      ;FOLD -- Hilfsflag SK Programmwechsel -- ;%{SE}%MKUKATPVW %CVW_COM %VCOMMENT %P 2:-- Hilfsflag SK Programmwechsel --, 3: VW_COMMENT
      ;ENDFOLD
      ;FOLD F334 = AUS ;%{SE}%MKUKATPVW %CVW_SPS %VBOASG %P 2:F334 = AUS, 3: BOASG
         $FLAG[334] = FALSE
      ;ENDFOLD
      ;FOLD A757 = F830 & A757 ;%{SE}%MKUKATPVW %CVW_SPS %VBOASG %P 2:A757 = F830 & A757, 3: BOASG
         $OUT[757] = $FLAG[830] AND $OUT[757]
      ;ENDFOLD
      ;FOLD -- EZ1/SP1 schliessen -- ;%{SE}%MKUKATPVW %CVW_COM %VCOMMENT %P 2:-- EZ1/SP1 schliessen --, 3: VW_COMMENT
      ;ENDFOLD
      ;FOLD A725 = !F830 & A725 ;%{SE}%MKUKATPVW %CVW_SPS %VBOASG %P 2:A725 = !F830 & A725, 3: BOASG
         $OUT[725] = NOT $FLAG[830] AND $OUT[725]
      ;ENDFOLD
      ;FOLD A717 = AUS ;%{SE}%MKUKATPVW %CVW_SPS %VBOASG %P 2:A717 = AUS, 3: BOASG
         $OUT[717] = FALSE
      ;ENDFOLD
      ;FOLD A718 = !F329 & !F122 ;%{SE}%MKUKATPVW %CVW_SPS %VBOASG %P 2:A718 = !F329 & !F122, 3: BOASG
         $OUT[718] = NOT $FLAG[329] AND NOT $FLAG[122]
      ;ENDFOLD
      ;FOLD -- Ueberwachungszeit Kurzschlussschweissung SK1 -- ;%{SE}%MKUKATPVW %CVW_COM %VCOMMENT %P 2:-- Ueberwachungszeit Kurzschlussschweissung SK1 --, 3: VW_COMMENT
      ;ENDFOLD
      ;FOLD t9 ( EIN ) = -80[1/10Sek] ;%{SE}%MKUKATPVW %CVW_SPS %VTASG %P 2:t9 ( EIN ) = -80[1/10Sek], 3: TASG
         VW(#SET_TIME,TRUE,9,0,-80)
      ;ENDFOLD
      ;FOLD Schritt 71 = T8 & !E717 & E718 + E717 & !E718 & (F329 + F326 + F122) & A4039  ;%{SE}%MKUKATPVW %CVW_SPS %VST_CON %P 2:Schritt 71 = T8 & !E717 & E718 + E717 & !E718 & (F329 + F326 + F122) & A4039 , 3: ST_CON
         IF $TIMER_FLAG[8] AND NOT $IN[717] AND $IN[718] OR $IN[717] AND NOT $IN[718] AND ($FLAG[329] OR $FLAG[326] OR $FLAG[122]) AND $OUT[4039] THEN
            PREVSTEP = $APP_INT[5]
            $APP_INT[5] = 71
         ENDIF
      ;ENDFOLD
   ;ENDFOLD
   ;FOLD SCHRITT 71 -- STAT EZ1/SP1/KE1-- ;%{P}%MKUKATPVW,%CSTEP,%VST_NR,%P 1:SCHRITT, 2:71, 3: STAT EZ1/SP1/KE1
      ;FOLD ;%{H}
         Case 71
      ;ENDFOLD
      ;FOLD -- Hilfsflag SK Programmwechsel -- ;%{SE}%MKUKATPVW %CVW_COM %VCOMMENT %P 2:-- Hilfsflag SK Programmwechsel --, 3: VW_COMMENT
      ;ENDFOLD
      ;FOLD F334 = AUS ;%{SE}%MKUKATPVW %CVW_SPS %VBOASG %P 2:F334 = AUS, 3: BOASG
         $FLAG[334] = FALSE
      ;ENDFOLD
      ;FOLD t9 ( EIN ) = STOP ;%{SE}%MKUKATPVW %CVW_SPS %VTSTOP %P 2:t9 ( EIN ) = STOP, 3: TSTOP
         VW(#SET_TIME,TRUE,9,1,0)
      ;ENDFOLD
      ;FOLD -- RSK Fehlerausgabe Kraftaufbau -- ;%{SE}%MKUKATPVW %CVW_COM %VCOMMENT %P 2:-- RSK Fehlerausgabe Kraftaufbau --, 3: VW_COMMENT
      ;ENDFOLD
      ;FOLD F325 = T9 + F325 ;%{SE}%MKUKATPVW %CVW_SPS %VBOASG %P 2:F325 = T9 + F325, 3: BOASG
         $FLAG[325] = $TIMER_FLAG[9] OR $FLAG[325]
      ;ENDFOLD
      ;FOLD -- RSK Fehlerausgabe K -- ;%{SE}%MKUKATPVW %CVW_COM %VCOMMENT %P 2:-- RSK Fehlerausgabe K --, 3: VW_COMMENT
      ;ENDFOLD
      ;FOLD F836 = (A718 & E788 + A718 & !E705) & F830 ;%{SE}%MKUKATPVW %CVW_SPS %VBOASG %P 2:F836 = (A718 & E788 + A718 & !E705) & F830, 3: BOASG
         $FLAG[836] = ($OUT[718] AND $IN[788] OR $OUT[718] AND NOT $IN[705]) AND $FLAG[830]
      ;ENDFOLD
      ;FOLD F327 = (A785 & E805 + A785 & !E802) &!F830 + F836 + F327 ;%{SE}%MKUKATPVW %CVW_SPS %VBOASG %P 2:F327 = (A785 & E805 + A785 & !E802) &!F830 + F836 + F327, 3: BOASG
         $FLAG[327] = ($OUT[785] AND $IN[805] OR $OUT[785] AND NOT $IN[802]) AND NOT $FLAG[830] OR $FLAG[836] OR $FLAG[327]
      ;ENDFOLD
      ;FOLD -- RSK Sammelstoerung -- ;%{SE}%MKUKATPVW %CVW_COM %VCOMMENT %P 2:-- RSK Sammelstoerung --, 3: VW_COMMENT
      ;ENDFOLD
      ;FOLD F329 = F325 + F326 + F327 ;%{SE}%MKUKATPVW %CVW_SPS %VBOASG %P 2:F329 = F325 + F326 + F327, 3: BOASG
         $FLAG[329] = $FLAG[325] OR $FLAG[326] OR $FLAG[327]
      ;ENDFOLD
      ;FOLD -- Kurzschlussschweissung SK1 -- ;%{SE}%MKUKATPVW %CVW_COM %VCOMMENT %P 2:-- Kurzschlussschweissung SK1 --, 3: VW_COMMENT
      ;ENDFOLD
      ;FOLD A785 = (!F325 & !F329 & !F122 & !F830) + (F830 & A785) ;%{SE}%MKUKATPVW %CVW_SPS %VBOASG %P 2:A785 = (!F325 & !F329 & !F122 & !F830) + (F830 & A785), 3: BOASG
         $OUT[785] = (NOT $FLAG[325] AND NOT $FLAG[329] AND NOT $FLAG[122] AND NOT $FLAG[830]) OR ($FLAG[830] AND $OUT[785])
      ;ENDFOLD
      ;FOLD F836 = AUS ;%{SE}%MKUKATPVW %CVW_SPS %VBOASG %P 2:F836 = AUS, 3: BOASG
         $FLAG[836] = FALSE
      ;ENDFOLD
      ;FOLD F836 = (E719 & E787 & !E789 + E719 & E15 + F326 + F327 + F122) & F830 & A4039 ;%{SE}%MKUKATPVW %CVW_SPS %VBOASG %P 2:F836 = (E719 & E787 & !E789 + E719 & E15 + F326 + F327 + F122) & F830 & A4039, 3: BOASG
         $FLAG[836] = ($IN[719] AND $IN[787] AND NOT $IN[789] OR $IN[719] AND $IN[15] OR $FLAG[326] OR $FLAG[327] OR $FLAG[122]) AND $FLAG[830] AND $OUT[4039]
      ;ENDFOLD
      ;FOLD -- Flagbildung Wiederholfraesen -- ;%{SE}%MKUKATPVW %CVW_COM %VCOMMENT %P 2:-- Flagbildung Wiederholfraesen --, 3: VW_COMMENT
      ;ENDFOLD
      ;FOLD F749 = (F322 + F323 + F325 + F326 + F327 + F329) & !F748 ;%{SE}%MKUKATPVW %CVW_SPS %VBOASG %P 2:F749 = (F322 + F323 + F325 + F326 + F327 + F329) & !F748, 3: BOASG
         $FLAG[749] = ($FLAG[322] OR $FLAG[323] OR $FLAG[325] OR $FLAG[326] OR $FLAG[327] OR $FLAG[329]) AND NOT $FLAG[748]
      ;ENDFOLD
      ;FOLD Schritt 72 = (E785 & E804 & !E806 + E785 & E15 + F326 + F327 + F122) & !F830 & A4039 + F836  ;%{SE}%MKUKATPVW %CVW_SPS %VST_CON %P 2:Schritt 72 = (E785 & E804 & !E806 + E785 & E15 + F326 + F327 + F122) & !F830 & A4039 + F836 , 3: ST_CON
         IF ($IN[785] AND $IN[804] AND NOT $IN[806] OR $IN[785] AND $IN[15] OR $FLAG[326] OR $FLAG[327] OR $FLAG[122]) AND NOT $FLAG[830] AND $OUT[4039] OR $FLAG[836] THEN
            PREVSTEP = $APP_INT[5]
            $APP_INT[5] = 72
         ENDIF
      ;ENDFOLD
   ;ENDFOLD
   ;FOLD SCHRITT 72 -- STAT EZ1/SP1/KE1 -- ;%{P}%MKUKATPVW,%CSTEP,%VST_NR,%P 1:SCHRITT, 2:72, 3: STAT EZ1/SP1/KE1
      ;FOLD ;%{H}
         Case 72
      ;ENDFOLD
      ;FOLD A785 = F830 & A785 ;%{SE}%MKUKATPVW %CVW_SPS %VBOASG %P 2:A785 = F830 & A785, 3: BOASG
         $OUT[785] = $FLAG[830] AND $OUT[785]
      ;ENDFOLD
      ;FOLD F78 = !F327 & F78 ;%{SE}%MKUKATPVW %CVW_SPS %VBOASG %P 2:F78 = !F327 & F78, 3: BOASG
         $FLAG[78] = NOT $FLAG[327] AND $FLAG[78]
      ;ENDFOLD
      ;FOLD F79 = F327 + F79 ;%{SE}%MKUKATPVW %CVW_SPS %VBOASG %P 2:F79 = F327 + F79, 3: BOASG
         $FLAG[79] = $FLAG[327] OR $FLAG[79]
      ;ENDFOLD
      ;FOLD F836 = AUS ;%{SE}%MKUKATPVW %CVW_SPS %VBOASG %P 2:F836 = AUS, 3: BOASG
         $FLAG[836] = FALSE
      ;ENDFOLD
      ;FOLD -- EZ1/SP1/KE1 SZ1 oeffnen -- ;%{SE}%MKUKATPVW %CVW_COM %VCOMMENT %P 2:-- EZ1/SP1/KE1 SZ1 oeffnen --, 3: VW_COMMENT
      ;ENDFOLD
      ;FOLD A719 = AUS ;%{SE}%MKUKATPVW %CVW_SPS %VBOASG %P 2:A719 = AUS, 3: BOASG
         $OUT[719] = FALSE
      ;ENDFOLD
      ;FOLD A718 = AUS ;%{SE}%MKUKATPVW %CVW_SPS %VBOASG %P 2:A718 = AUS, 3: BOASG
         $OUT[718] = FALSE
      ;ENDFOLD
      ;FOLD A717 = !E717 ;%{SE}%MKUKATPVW %CVW_SPS %VBOASG %P 2:A717 = !E717, 3: BOASG
         $OUT[717] = NOT $IN[717]
      ;ENDFOLD
      ;FOLD F836 = !F326 & !F830 ;%{SE}%MKUKATPVW %CVW_SPS %VBOASG %P 2:F836 = !F326 & !F830, 3: BOASG
         $FLAG[836] = NOT $FLAG[326] AND NOT $FLAG[830]
      ;ENDFOLD
      ;FOLD bin3 ( F836 ) = 1 ;%{SE}%MKUKATPVW %CVW_SPS %VARIASG %P 2:bin3 ( F836 ) = 1, 3: ARIASG
         VW(#BINOUT,$FLAG[836],3,1)
      ;ENDFOLD
      ;FOLD -- Wartezeit Programmwechsel SK -- ;%{SE}%MKUKATPVW %CVW_COM %VCOMMENT %P 2:-- Wartezeit Programmwechsel SK --, 3: VW_COMMENT
      ;ENDFOLD
      ;FOLD T8 ( !F334 ) = -2[1/10Sek] ;%{SE}%MKUKATPVW %CVW_SPS %VTASG %P 2:T8 ( !F334 ) = -2[1/10Sek], 3: TASG
         VW(#SET_TIME,NOT $FLAG[334],8,0,-2)
      ;ENDFOLD
      ;FOLD -- Hilfsflag SK Programmwechsel -- ;%{SE}%MKUKATPVW %CVW_COM %VCOMMENT %P 2:-- Hilfsflag SK Programmwechsel --, 3: VW_COMMENT
      ;ENDFOLD
      ;FOLD F334 = EIN ;%{SE}%MKUKATPVW %CVW_SPS %VBOASG %P 2:F334 = EIN, 3: BOASG
         $FLAG[334] = TRUE
      ;ENDFOLD
      ;FOLD F748 = F322 + F323 + F325 + F326 + F327 + F329 ;%{SE}%MKUKATPVW %CVW_SPS %VBOASG %P 2:F748 = F322 + F323 + F325 + F326 + F327 + F329, 3: BOASG
         $FLAG[748] = $FLAG[322] OR $FLAG[323] OR $FLAG[325] OR $FLAG[326] OR $FLAG[327] OR $FLAG[329]
      ;ENDFOLD
      ;FOLD Schritt 51 = E717 & !E718 & (F322 + F323 + F325 + F326 + F327 + F329) & (E26 + E27) & A4039  ;%{SE}%MKUKATPVW %CVW_SPS %VST_CON %P 2:Schritt 51 = E717 & !E718 & (F322 + F323 + F325 + F326 + F327 + F329) & (E26 + E27) & A4039 , 3: ST_CON
         IF $IN[717] AND NOT $IN[718] AND ($FLAG[322] OR $FLAG[323] OR $FLAG[325] OR $FLAG[326] OR $FLAG[327] OR $FLAG[329]) AND ($IN[26] OR $IN[27]) AND $OUT[4039] THEN
            PREVSTEP = $APP_INT[5]
            $APP_INT[5] = 51
         ENDIF
      ;ENDFOLD
      ;FOLD Schritt 51 = E717 & !E718 & (F322 + F323 + F325 + F326 + F327 + F329) & (F749 & F731) & A4039  ;%{SE}%MKUKATPVW %CVW_SPS %VST_CON %P 2:Schritt 51 = E717 & !E718 & (F322 + F323 + F325 + F326 + F327 + F329) & (F749 & F731) & A4039 , 3: ST_CON
         IF $IN[717] AND NOT $IN[718] AND ($FLAG[322] OR $FLAG[323] OR $FLAG[325] OR $FLAG[326] OR $FLAG[327] OR $FLAG[329]) AND ($FLAG[749] AND $FLAG[731]) AND $OUT[4039] THEN
            PREVSTEP = $APP_INT[5]
            $APP_INT[5] = 51
         ENDIF
      ;ENDFOLD
      ;FOLD Schritt 73 = T8 & E717 & !E718 & (!F325 & !F326 & !F327 & !F329 + F122) & A4039  ;%{SE}%MKUKATPVW %CVW_SPS %VST_CON %P 2:Schritt 73 = T8 & E717 & !E718 & (!F325 & !F326 & !F327 & !F329 + F122) & A4039 , 3: ST_CON
         IF $TIMER_FLAG[8] AND $IN[717] AND NOT $IN[718] AND (NOT $FLAG[325] AND NOT $FLAG[326] AND NOT $FLAG[327] AND NOT $FLAG[329] OR $FLAG[122]) AND $OUT[4039] THEN
            PREVSTEP = $APP_INT[5]
            $APP_INT[5] = 73
         ENDIF
      ;ENDFOLD
   ;ENDFOLD
   ;FOLD SCHRITT 73 -- STAT EZ1/SP1/KE1 # Ende -- ;%{P}%MKUKATPVW,%CSTEP,%VST_NR,%P 1:SCHRITT, 2:73, 3: STAT EZ1/SP1/KE1 # Ende
      ;FOLD ;%{H}
         Case 73
      ;ENDFOLD
      ;FOLD -- Hilfsflag SK Programmwechsel -- ;%{SE}%MKUKATPVW %CVW_COM %VCOMMENT %P 2:-- Hilfsflag SK Programmwechsel --, 3: VW_COMMENT
      ;ENDFOLD
      ;FOLD F334 = AUS ;%{SE}%MKUKATPVW %CVW_SPS %VBOASG %P 2:F334 = AUS, 3: BOASG
         $FLAG[334] = FALSE
      ;ENDFOLD
      ;FOLD A116 = AUS ;%{SE}%MKUKATPVW %CVW_SPS %VBOASG %P 2:A116 = AUS, 3: BOASG
         $OUT[116] = FALSE
      ;ENDFOLD
      ;FOLD A130 = AUS ;%{SE}%MKUKATPVW %CVW_SPS %VBOASG %P 2:A130 = AUS, 3: BOASG
         $OUT[130] = FALSE
      ;ENDFOLD
      ;FOLD F836 = AUS ;%{SE}%MKUKATPVW %CVW_SPS %VBOASG %P 2:F836 = AUS, 3: BOASG
         $FLAG[836] = FALSE
      ;ENDFOLD
      ;FOLD -- RSK Sammelstoerung -- ;%{SE}%MKUKATPVW %CVW_COM %VCOMMENT %P 2:-- RSK Sammelstoerung --, 3: VW_COMMENT
      ;ENDFOLD
      ;FOLD F329 = F122 ;%{SE}%MKUKATPVW %CVW_SPS %VBOASG %P 2:F329 = F122, 3: BOASG
         $FLAG[329] = $FLAG[122]
      ;ENDFOLD
      ;FOLD F93 = (!E786 & E787 & !E788 & !F830) + (!E721 & !E723 & E724 & F830) + F122 & (E26 + E27) ;%{SE}%MKUKATPVW %CVW_SPS %VBOASG %P 2:F93 = (!E786 & E787 & !E788 & !F830) + (!E721 & !E723 & E724 & F830) + F122 & (E26 + E27), 3: BOASG
         $FLAG[93] = (NOT $IN[786] AND $IN[787] AND NOT $IN[788] AND NOT $FLAG[830]) OR (NOT $IN[721] AND NOT $IN[723] AND $IN[724] AND $FLAG[830]) OR $FLAG[122] AND ($IN[26] OR $IN[27])
      ;ENDFOLD
      ;FOLD Schritt 1 = F93 & A4039  ;%{SE}%MKUKATPVW %CVW_SPS %VST_CON %P 2:Schritt 1 = F93 & A4039 , 3: ST_CON
         IF $FLAG[93] AND $OUT[4039] THEN
            PREVSTEP = $APP_INT[5]
            $APP_INT[5] = 1
         ENDIF
      ;ENDFOLD
   ;ENDFOLD
   ;FOLD SCHRITT 74 -- STAT EZ2/SP2/KE2 # Start-- ;%{P}%MKUKATPVW,%CSTEP,%VST_NR,%P 1:SCHRITT, 2:74, 3: STAT EZ2/SP2/KE2 # Start
      ;FOLD ;%{H}
         Case 74
      ;ENDFOLD
      ;FOLD -- RSK gestartet -- ;%{SE}%MKUKATPVW %CVW_COM %VCOMMENT %P 2:-- RSK gestartet --, 3: VW_COMMENT
      ;ENDFOLD
      ;FOLD F160 = AUS ;%{SE}%MKUKATPVW %CVW_SPS %VBOASG %P 2:F160 = AUS, 3: BOASG
         $FLAG[160] = FALSE
      ;ENDFOLD
      ;FOLD F321 = AUS ;%{SE}%MKUKATPVW %CVW_SPS %VBOASG %P 2:F321 = AUS, 3: BOASG
         $FLAG[321] = FALSE
      ;ENDFOLD
      ;FOLD F322 = AUS ;%{SE}%MKUKATPVW %CVW_SPS %VBOASG %P 2:F322 = AUS, 3: BOASG
         $FLAG[322] = FALSE
      ;ENDFOLD
      ;FOLD F323 = AUS ;%{SE}%MKUKATPVW %CVW_SPS %VBOASG %P 2:F323 = AUS, 3: BOASG
         $FLAG[323] = FALSE
      ;ENDFOLD
      ;FOLD F324 = AUS ;%{SE}%MKUKATPVW %CVW_SPS %VBOASG %P 2:F324 = AUS, 3: BOASG
         $FLAG[324] = FALSE
      ;ENDFOLD
      ;FOLD F325 = AUS ;%{SE}%MKUKATPVW %CVW_SPS %VBOASG %P 2:F325 = AUS, 3: BOASG
         $FLAG[325] = FALSE
      ;ENDFOLD
      ;FOLD F326 = AUS ;%{SE}%MKUKATPVW %CVW_SPS %VBOASG %P 2:F326 = AUS, 3: BOASG
         $FLAG[326] = FALSE
      ;ENDFOLD
      ;FOLD F327 = AUS ;%{SE}%MKUKATPVW %CVW_SPS %VBOASG %P 2:F327 = AUS, 3: BOASG
         $FLAG[327] = FALSE
      ;ENDFOLD
      ;FOLD F329 = AUS ;%{SE}%MKUKATPVW %CVW_SPS %VBOASG %P 2:F329 = AUS, 3: BOASG
         $FLAG[329] = FALSE
      ;ENDFOLD
      ;FOLD -- EZ2/SP2/KE2 Zaehler -- ;%{SE}%MKUKATPVW %CVW_COM %VCOMMENT %P 2:-- EZ2/SP2/KE2 Zaehler --, 3: VW_COMMENT
      ;ENDFOLD
      ;FOLD F150 = AUS ;%{SE}%MKUKATPVW %CVW_SPS %VBOASG %P 2:F150 = AUS, 3: BOASG
         $FLAG[150] = FALSE
      ;ENDFOLD
      ;FOLD F151 = AUS ;%{SE}%MKUKATPVW %CVW_SPS %VBOASG %P 2:F151 = AUS, 3: BOASG
         $FLAG[151] = FALSE
      ;ENDFOLD
      ;FOLD F152 = AUS ;%{SE}%MKUKATPVW %CVW_SPS %VBOASG %P 2:F152 = AUS, 3: BOASG
         $FLAG[152] = FALSE
      ;ENDFOLD
      ;FOLD F153 = AUS ;%{SE}%MKUKATPVW %CVW_SPS %VBOASG %P 2:F153 = AUS, 3: BOASG
         $FLAG[153] = FALSE
      ;ENDFOLD
      ;FOLD F154 = AUS ;%{SE}%MKUKATPVW %CVW_SPS %VBOASG %P 2:F154 = AUS, 3: BOASG
         $FLAG[154] = FALSE
      ;ENDFOLD
      ;FOLD F155 = AUS ;%{SE}%MKUKATPVW %CVW_SPS %VBOASG %P 2:F155 = AUS, 3: BOASG
         $FLAG[155] = FALSE
      ;ENDFOLD
      ;FOLD -- Hilfsflags Funktionstest KF Motor -- ;%{SE}%MKUKATPVW %CVW_COM %VCOMMENT %P 2:-- Hilfsflags Funktionstest KF Motor --, 3: VW_COMMENT
      ;ENDFOLD
      ;FOLD F312 = AUS ;%{SE}%MKUKATPVW %CVW_SPS %VBOASG %P 2:F312 = AUS, 3: BOASG
         $FLAG[312] = FALSE
      ;ENDFOLD
      ;FOLD F313 = AUS ;%{SE}%MKUKATPVW %CVW_SPS %VBOASG %P 2:F313 = AUS, 3: BOASG
         $FLAG[313] = FALSE
      ;ENDFOLD
      ;FOLD bin3 ( F285 ) = 35 ;%{SE}%MKUKATPVW %CVW_SPS %VARIASG %P 2:bin3 ( F285 ) = 35, 3: ARIASG
         VW(#BINOUT,$FLAG[285],3,35)
      ;ENDFOLD
      ;FOLD bin4 ( EIN ) = 31 ;%{SE}%MKUKATPVW %CVW_SPS %VARIASG %P 2:bin4 ( EIN ) = 31, 3: ARIASG
         VW(#BINOUT,TRUE,4,31)
      ;ENDFOLD
      ;FOLD bin6 ( !F285 ) = 31 ;%{SE}%MKUKATPVW %CVW_SPS %VARIASG %P 2:bin6 ( !F285 ) = 31, 3: ARIASG
         VW(#BINOUT,NOT $FLAG[285],6,31)
      ;ENDFOLD
      ;FOLD -- Wartezeit Programmwechsel SK -- ;%{SE}%MKUKATPVW %CVW_COM %VCOMMENT %P 2:-- Wartezeit Programmwechsel SK --, 3: VW_COMMENT
      ;ENDFOLD
      ;FOLD T8 ( !F334 ) = -2[1/10Sek] ;%{SE}%MKUKATPVW %CVW_SPS %VTASG %P 2:T8 ( !F334 ) = -2[1/10Sek], 3: TASG
         VW(#SET_TIME,NOT $FLAG[334],8,0,-2)
      ;ENDFOLD
      ;FOLD -- Hilfsflag SK Programmwechsel -- ;%{SE}%MKUKATPVW %CVW_COM %VCOMMENT %P 2:-- Hilfsflag SK Programmwechsel --, 3: VW_COMMENT
      ;ENDFOLD
      ;FOLD F334 = EIN ;%{SE}%MKUKATPVW %CVW_SPS %VBOASG %P 2:F334 = EIN, 3: BOASG
         $FLAG[334] = TRUE
      ;ENDFOLD
      ;FOLD -- Stat. EZ2/SP2/KE2 beim Fraesen -- ;%{SE}%MKUKATPVW %CVW_COM %VCOMMENT %P 2:-- Stat. EZ2/SP2/KE2 beim Fraesen --, 3: VW_COMMENT
      ;ENDFOLD
      ;FOLD A116 = EIN ;%{SE}%MKUKATPVW %CVW_SPS %VBOASG %P 2:A116 = EIN, 3: BOASG
         $OUT[116] = TRUE
      ;ENDFOLD
      ;FOLD A162 = EIN ;%{SE}%MKUKATPVW %CVW_SPS %VBOASG %P 2:A162 = EIN, 3: BOASG
         $OUT[162] = TRUE
      ;ENDFOLD
      ;FOLD -- Quitt. Fraesen SK1 AUS -- ;%{SE}%MKUKATPVW %CVW_COM %VCOMMENT %P 2:-- Quitt. Fraesen SK1 AUS --, 3: VW_COMMENT
      ;ENDFOLD
      ;FOLD A786 = F830 ;%{SE}%MKUKATPVW %CVW_SPS %VBOASG %P 2:A786 = F830, 3: BOASG
         $OUT[786] = $FLAG[830]
      ;ENDFOLD
      ;FOLD A722 = !F830 ;%{SE}%MKUKATPVW %CVW_SPS %VBOASG %P 2:A722 = !F830, 3: BOASG
         $OUT[722] = NOT $FLAG[830]
      ;ENDFOLD
      ;FOLD -- Quitt. Fraesen SK2 AUS -- ;%{SE}%MKUKATPVW %CVW_COM %VCOMMENT %P 2:-- Quitt. Fraesen SK2 AUS --, 3: VW_COMMENT
      ;ENDFOLD
      ;FOLD A946 = F831 & A946 ;%{SE}%MKUKATPVW %CVW_SPS %VBOASG %P 2:A946 = F831 & A946, 3: BOASG
         $OUT[946] = $FLAG[831] AND $OUT[946]
      ;ENDFOLD
      ;FOLD A882 = !F831 & A882 ;%{SE}%MKUKATPVW %CVW_SPS %VBOASG %P 2:A882 = !F831 & A882, 3: BOASG
         $OUT[882] = NOT $FLAG[831] AND $OUT[882]
      ;ENDFOLD
      ;FOLD Schritt 75 = T8 & A4039  ;%{SE}%MKUKATPVW %CVW_SPS %VST_CON %P 2:Schritt 75 = T8 & A4039 , 3: ST_CON
         IF $TIMER_FLAG[8] AND $OUT[4039] THEN
            PREVSTEP = $APP_INT[5]
            $APP_INT[5] = 75
         ENDIF
      ;ENDFOLD
   ;ENDFOLD
   ;FOLD SCHRITT 75 -- STAT EZ2/SP2/KE2 -- ;%{P}%MKUKATPVW,%CSTEP,%VST_NR,%P 1:SCHRITT, 2:75, 3: STAT EZ2/SP2/KE2
      ;FOLD ;%{H}
         Case 75
      ;ENDFOLD
      ;FOLD -- Hilfsflag SK Programmwechsel -- ;%{SE}%MKUKATPVW %CVW_COM %VCOMMENT %P 2:-- Hilfsflag SK Programmwechsel --, 3: VW_COMMENT
      ;ENDFOLD
      ;FOLD F334 = AUS ;%{SE}%MKUKATPVW %CVW_SPS %VBOASG %P 2:F334 = AUS, 3: BOASG
         $FLAG[334] = FALSE
      ;ENDFOLD
      ;FOLD -- Ueberwachungszeit KF2 EIN -- ;%{SE}%MKUKATPVW %CVW_COM %VCOMMENT %P 2:-- Ueberwachungszeit KF2 EIN --, 3: VW_COMMENT
      ;ENDFOLD
      ;FOLD T7 ( EIN ) = -50[1/10Sek] ;%{SE}%MKUKATPVW %CVW_SPS %VTASG %P 2:T7 ( EIN ) = -50[1/10Sek], 3: TASG
         VW(#SET_TIME,TRUE,7,0,-50)
      ;ENDFOLD
      ;FOLD -- KF2 einschalten -- ;%{SE}%MKUKATPVW %CVW_COM %VCOMMENT %P 2:-- KF2 einschalten --, 3: VW_COMMENT
      ;ENDFOLD
      ;FOLD i1 (EIN) = 0 ;%{SE}%MKUKATPVW %CVW_SPS %VARIASG %P 2:i1 (EIN) = 0, 3: ARIASG
         VW(#COUNTER,TRUE,1,0)
      ;ENDFOLD
      ;FOLD A994 = EIN ;%{SE}%MKUKATPVW %CVW_SPS %VBOASG %P 2:A994 = EIN, 3: BOASG
         $OUT[994] = TRUE
      ;ENDFOLD
      ;FOLD Schritt 76 = A4039  ;%{SE}%MKUKATPVW %CVW_SPS %VST_CON %P 2:Schritt 76 = A4039 , 3: ST_CON
         IF $OUT[4039] THEN
            PREVSTEP = $APP_INT[5]
            $APP_INT[5] = 76
         ENDIF
      ;ENDFOLD
   ;ENDFOLD
   ;FOLD SCHRITT 76 -- STAT EZ2/SP2/KE2 -- ;%{P}%MKUKATPVW,%CSTEP,%VST_NR,%P 1:SCHRITT, 2:76, 3: STAT EZ2/SP2/KE2
      ;FOLD ;%{H}
         Case 76
      ;ENDFOLD
      ;FOLD -- Funktionstest KF Motor -- ;%{SE}%MKUKATPVW %CVW_COM %VCOMMENT %P 2:-- Funktionstest KF Motor --, 3: VW_COMMENT
      ;ENDFOLD
      ;FOLD F312 = EIN ;%{SE}%MKUKATPVW %CVW_SPS %VBOASG %P 2:F312 = EIN, 3: BOASG
         $FLAG[312] = TRUE
      ;ENDFOLD
      ;FOLD F313 = i1 > 2 ;%{SE}%MKUKATPVW %CVW_SPS %VBOCMP %P 2:F313 = i1 > 2, 3: BOCMP
         $FLAG[313] = $COUNT_I[1] > 2
      ;ENDFOLD
      ;FOLD Schritt 77 = (F313 + T7) & A4039  ;%{SE}%MKUKATPVW %CVW_SPS %VST_CON %P 2:Schritt 77 = (F313 + T7) & A4039 , 3: ST_CON
         IF ($FLAG[313] OR $TIMER_FLAG[7]) AND $OUT[4039] THEN
            PREVSTEP = $APP_INT[5]
            $APP_INT[5] = 77
         ENDIF
      ;ENDFOLD
   ;ENDFOLD
   ;FOLD SCHRITT 77 -- STAT EZ2/SP2/KE2-- ;%{P}%MKUKATPVW,%CSTEP,%VST_NR,%P 1:SCHRITT, 2:77, 3: STAT EZ2/SP2/KE2
      ;FOLD ;%{H}
         Case 77
      ;ENDFOLD
      ;FOLD F312 = AUS ;%{SE}%MKUKATPVW %CVW_SPS %VBOASG %P 2:F312 = AUS, 3: BOASG
         $FLAG[312] = FALSE
      ;ENDFOLD
      ;FOLD -- Ueberwachungszeit KS2 schwenken -- ;%{SE}%MKUKATPVW %CVW_COM %VCOMMENT %P 2:-- Ueberwachungszeit KS2 schwenken --, 3: VW_COMMENT
      ;ENDFOLD
      ;FOLD t8 ( EIN ) = -100[1/10Sek] ;%{SE}%MKUKATPVW %CVW_SPS %VTASG %P 2:t8 ( EIN ) = -100[1/10Sek], 3: TASG
         VW(#SET_TIME,TRUE,8,0,-100)
      ;ENDFOLD
      ;FOLD Schritt 78 = A4039  ;%{SE}%MKUKATPVW %CVW_SPS %VST_CON %P 2:Schritt 78 = A4039 , 3: ST_CON
         IF $OUT[4039] THEN
            PREVSTEP = $APP_INT[5]
            $APP_INT[5] = 78
         ENDIF
      ;ENDFOLD
   ;ENDFOLD
   ;FOLD SCHRITT 78 -- STAT EZ2/SP2/KE2 -- ;%{P}%MKUKATPVW,%CSTEP,%VST_NR,%P 1:SCHRITT, 2:78, 3: STAT EZ2/SP2/KE2
      ;FOLD ;%{H}
         Case 78
      ;ENDFOLD
      ;FOLD -- RSK Fehlerausgabe KF1 Initiator/Motor -- ;%{SE}%MKUKATPVW %CVW_COM %VCOMMENT %P 2:-- RSK Fehlerausgabe KF1 Initiator/Motor --, 3: VW_COMMENT
      ;ENDFOLD
      ;FOLD F322 = !F313 ;%{SE}%MKUKATPVW %CVW_SPS %VBOASG %P 2:F322 = !F313, 3: BOASG
         $FLAG[322] = NOT $FLAG[313]
      ;ENDFOLD
      ;FOLD -- RSK Fehlerausgabe KS2 Ruhest. -- ;%{SE}%MKUKATPVW %CVW_COM %VCOMMENT %P 2:-- RSK Fehlerausgabe KS2 Ruhest. --, 3: VW_COMMENT
      ;ENDFOLD
      ;FOLD F323 = (!E1002 + E1003 + E1004 + !E1005) & !F324 & !F328 ;%{SE}%MKUKATPVW %CVW_SPS %VBOASG %P 2:F323 = (!E1002 + E1003 + E1004 + !E1005) & !F324 & !F328, 3: BOASG
         $FLAG[323] = (NOT $IN[1002] OR $IN[1003] OR $IN[1004] OR NOT $IN[1005]) AND NOT $FLAG[324] AND NOT $FLAG[328]
      ;ENDFOLD
      ;FOLD -- RSK Sammelstoerung -- ;%{SE}%MKUKATPVW %CVW_COM %VCOMMENT %P 2:-- RSK Sammelstoerung --, 3: VW_COMMENT
      ;ENDFOLD
      ;FOLD F329 = F322 + F323 ;%{SE}%MKUKATPVW %CVW_SPS %VBOASG %P 2:F329 = F322 + F323, 3: BOASG
         $FLAG[329] = $FLAG[322] OR $FLAG[323]
      ;ENDFOLD
      ;FOLD T7 ( EIN ) = STOP ;%{SE}%MKUKATPVW %CVW_SPS %VTSTOP %P 2:T7 ( EIN ) = STOP, 3: TSTOP
         VW(#SET_TIME,TRUE,7,1,0)
      ;ENDFOLD
      ;FOLD A994 = !F322 & !F323 ;%{SE}%MKUKATPVW %CVW_SPS %VBOASG %P 2:A994 = !F322 & !F323, 3: BOASG
         $OUT[994] = NOT $FLAG[322] AND NOT $FLAG[323]
      ;ENDFOLD
      ;FOLD -- KF2 Versetzeinheit vor -- ;%{SE}%MKUKATPVW %CVW_COM %VCOMMENT %P 2:-- KF2 Versetzeinheit vor --, 3: VW_COMMENT
      ;ENDFOLD
      ;FOLD A995 = !F322 & !F323 & F564 ;%{SE}%MKUKATPVW %CVW_SPS %VBOASG %P 2:A995 = !F322 & !F323 & F564, 3: BOASG
         $OUT[995] = NOT $FLAG[322] AND NOT $FLAG[323] AND $FLAG[564]
      ;ENDFOLD
      ;FOLD Schritt 79 = (!F322 & !F323 & (E995 & F564 + !E995 & !F564) + T8) & A4039  ;%{SE}%MKUKATPVW %CVW_SPS %VST_CON %P 2:Schritt 79 = (!F322 & !F323 & (E995 & F564 + !E995 & !F564) + T8) & A4039 , 3: ST_CON
         IF (NOT $FLAG[322] AND NOT $FLAG[323] AND ($IN[995] AND $FLAG[564] OR NOT $IN[995] AND NOT $FLAG[564]) OR $TIMER_FLAG[8]) AND $OUT[4039] THEN
            PREVSTEP = $APP_INT[5]
            $APP_INT[5] = 79
         ENDIF
      ;ENDFOLD
      ;FOLD Schritt 95 = (F322 + F323) & !F324 & !F328 & A4039  ;%{SE}%MKUKATPVW %CVW_SPS %VST_CON %P 2:Schritt 95 = (F322 + F323) & !F324 & !F328 & A4039 , 3: ST_CON
         IF ($FLAG[322] OR $FLAG[323]) AND NOT $FLAG[324] AND NOT $FLAG[328] AND $OUT[4039] THEN
            PREVSTEP = $APP_INT[5]
            $APP_INT[5] = 95
         ENDIF
      ;ENDFOLD
   ;ENDFOLD
   ;FOLD SCHRITT 79 -- STAT EZ2/SP2/KE2 -- ;%{P}%MKUKATPVW,%CSTEP,%VST_NR,%P 1:SCHRITT, 2:79, 3: STAT EZ2/SP2/KE2
      ;FOLD ;%{H}
         Case 79
      ;ENDFOLD
      ;FOLD -- RSK Sammelstoerung -- ;%{SE}%MKUKATPVW %CVW_COM %VCOMMENT %P 2:-- RSK Sammelstoerung --, 3: VW_COMMENT
      ;ENDFOLD
      ;FOLD F329 = T8 ;%{SE}%MKUKATPVW %CVW_SPS %VBOASG %P 2:F329 = T8, 3: BOASG
         $FLAG[329] = $TIMER_FLAG[8]
      ;ENDFOLD
      ;FOLD F324 = AUS ;%{SE}%MKUKATPVW %CVW_SPS %VBOASG %P 2:F324 = AUS, 3: BOASG
         $FLAG[324] = FALSE
      ;ENDFOLD
      ;FOLD F328 = AUS ;%{SE}%MKUKATPVW %CVW_SPS %VBOASG %P 2:F328 = AUS, 3: BOASG
         $FLAG[328] = FALSE
      ;ENDFOLD
      ;FOLD -- KS2 in Arbeitsstellung schwenken -- ;%{SE}%MKUKATPVW %CVW_COM %VCOMMENT %P 2:-- KS2 in Arbeitsstellung schwenken --, 3: VW_COMMENT
      ;ENDFOLD
      ;FOLD A1002 = (F746 + !F714) & (E877 + F714) & !E1003 & (E995 & F564 + !E995 & !F564) ;%{SE}%MKUKATPVW %CVW_SPS %VBOASG %P 2:A1002 = (F746 + !F714) & (E877 + F714) & !E1003 & (E995 & F564 + !E995 & !F564), 3: BOASG
         $OUT[1002] = ($FLAG[746] OR NOT $FLAG[714]) AND ($IN[877] OR $FLAG[714]) AND NOT $IN[1003] AND ($IN[995] AND $FLAG[564] OR NOT $IN[995] AND NOT $FLAG[564])
      ;ENDFOLD
      ;FOLD -- KF2 Ausblasen -- ;%{SE}%MKUKATPVW %CVW_COM %VCOMMENT %P 2:-- KF2 Ausblasen --, 3: VW_COMMENT
      ;ENDFOLD
      ;FOLD A1007 = F330 + !F330 & !F331 & !F332 ;%{SE}%MKUKATPVW %CVW_SPS %VBOASG %P 2:A1007 = F330 + !F330 & !F331 & !F332, 3: BOASG
         $OUT[1007] = $FLAG[330] OR NOT $FLAG[330] AND NOT $FLAG[331] AND NOT $FLAG[332]
      ;ENDFOLD
      ;FOLD Schritt 80 = (F746 + !F714) & (E877 + F714) & (A1002 + E1003 + T8) & A4039  ;%{SE}%MKUKATPVW %CVW_SPS %VST_CON %P 2:Schritt 80 = (F746 + !F714) & (E877 + F714) & (A1002 + E1003 + T8) & A4039 , 3: ST_CON
         IF ($FLAG[746] OR NOT $FLAG[714]) AND ($IN[877] OR $FLAG[714]) AND ($OUT[1002] OR $IN[1003] OR $TIMER_FLAG[8]) AND $OUT[4039] THEN
            PREVSTEP = $APP_INT[5]
            $APP_INT[5] = 80
         ENDIF
      ;ENDFOLD
   ;ENDFOLD
   ;FOLD SCHRITT 80 -- STAT EZ2/SP2/KE2 -- ;%{P}%MKUKATPVW,%CSTEP,%VST_NR,%P 1:SCHRITT, 2:80, 3: STAT EZ2/SP2/KE2
      ;FOLD ;%{H}
         Case 80
      ;ENDFOLD
      ;FOLD -- RSK Fehlerausgabe KF Versetzeinheit -- ;%{SE}%MKUKATPVW %CVW_COM %VCOMMENT %P 2:-- RSK Fehlerausgabe KF Versetzeinheit --, 3: VW_COMMENT
      ;ENDFOLD
      ;FOLD F328 = !E995 & F564 & !F324 ;%{SE}%MKUKATPVW %CVW_SPS %VBOASG %P 2:F328 = !E995 & F564 & !F324, 3: BOASG
         $FLAG[328] = NOT $IN[995] AND $FLAG[564] AND NOT $FLAG[324]
      ;ENDFOLD
      ;FOLD -- RSK Fehlerausgabe KS2 Arbeitsstellung -- ;%{SE}%MKUKATPVW %CVW_COM %VCOMMENT %P 2:-- RSK Fehlerausgabe KS2 Arbeitsstellung --, 3: VW_COMMENT
      ;ENDFOLD
      ;FOLD F324 = (E1002 + !E1003 + !E1004 + E1005) & T8 & (E995 + !F564) + F324 ;%{SE}%MKUKATPVW %CVW_SPS %VBOASG %P 2:F324 = (E1002 + !E1003 + !E1004 + E1005) & T8 & (E995 + !F564) + F324, 3: BOASG
         $FLAG[324] = ($IN[1002] OR NOT $IN[1003] OR NOT $IN[1004] OR $IN[1005]) AND $TIMER_FLAG[8] AND ($IN[995] OR NOT $FLAG[564]) OR $FLAG[324]
      ;ENDFOLD
      ;FOLD -- RSK Fehlerausgabe EZ/SP min. Oeffnung -- ;%{SE}%MKUKATPVW %CVW_COM %VCOMMENT %P 2:-- RSK Fehlerausgabe EZ/SP min. Oeffnung --, 3: VW_COMMENT
      ;ENDFOLD
      ;FOLD F333 = !F746 ;%{SE}%MKUKATPVW %CVW_SPS %VBOASG %P 2:F333 = !F746, 3: BOASG
         $FLAG[333] = NOT $FLAG[746]
      ;ENDFOLD
      ;FOLD -- RSK Sammelstoerung -- ;%{SE}%MKUKATPVW %CVW_COM %VCOMMENT %P 2:-- RSK Sammelstoerung --, 3: VW_COMMENT
      ;ENDFOLD
      ;FOLD F329 = F324 + F328 + F333 ;%{SE}%MKUKATPVW %CVW_SPS %VBOASG %P 2:F329 = F324 + F328 + F333, 3: BOASG
         $FLAG[329] = $FLAG[324] OR $FLAG[328] OR $FLAG[333]
      ;ENDFOLD
      ;FOLD A994 = !F324 & !F328 ;%{SE}%MKUKATPVW %CVW_SPS %VBOASG %P 2:A994 = !F324 & !F328, 3: BOASG
         $OUT[994] = NOT $FLAG[324] AND NOT $FLAG[328]
      ;ENDFOLD
      ;FOLD -- KF1 Ausblasen -- ;%{SE}%MKUKATPVW %CVW_COM %VCOMMENT %P 2:-- KF1 Ausblasen --, 3: VW_COMMENT
      ;ENDFOLD
      ;FOLD A1007 = (F330 + !F330 & !F331 & !F332) & !F324 & !F328 ;%{SE}%MKUKATPVW %CVW_SPS %VBOASG %P 2:A1007 = (F330 + !F330 & !F331 & !F332) & !F324 & !F328, 3: BOASG
         $OUT[1007] = ($FLAG[330] OR NOT $FLAG[330] AND NOT $FLAG[331] AND NOT $FLAG[332]) AND NOT $FLAG[324] AND NOT $FLAG[328]
      ;ENDFOLD
      ;FOLD A995 = F564 ;%{SE}%MKUKATPVW %CVW_SPS %VBOASG %P 2:A995 = F564, 3: BOASG
         $OUT[995] = $FLAG[564]
      ;ENDFOLD
      ;FOLD -- Ueberwachungszeit EZ2/SP2/KE2 schliessen -- ;%{SE}%MKUKATPVW %CVW_COM %VCOMMENT %P 2:-- Ueberwachungszeit EZ2/SP2/KE2 schliessen --, 3: VW_COMMENT
      ;ENDFOLD
      ;FOLD t9 ( EIN ) = -80[1/10Sek] ;%{SE}%MKUKATPVW %CVW_SPS %VTASG %P 2:t9 ( EIN ) = -80[1/10Sek], 3: TASG
         VW(#SET_TIME,TRUE,9,0,-80)
      ;ENDFOLD
      ;FOLD -- Verweilzeit Versetzeinheit Rueck -- ;%{SE}%MKUKATPVW %CVW_COM %VCOMMENT %P 2:-- Verweilzeit Versetzeinheit Rueck --, 3: VW_COMMENT
      ;ENDFOLD
      ;FOLD t11 ( EIN ) = i24[1/10Sek] ;%{SE}%MKUKATPVW %CVW_SPS %VTASG %P 2:t11 ( EIN ) = i24[1/10Sek], 3: TASG
         VW(#SET_TIME,TRUE,11,0,$COUNT_I[24])
      ;ENDFOLD
      ;FOLD Schritt 75 = (F324 + F328) & (E26 + E27) & A4039  ;%{SE}%MKUKATPVW %CVW_SPS %VST_CON %P 2:Schritt 75 = (F324 + F328) & (E26 + E27) & A4039 , 3: ST_CON
         IF ($FLAG[324] OR $FLAG[328]) AND ($IN[26] OR $IN[27]) AND $OUT[4039] THEN
            PREVSTEP = $APP_INT[5]
            $APP_INT[5] = 75
         ENDIF
      ;ENDFOLD
      ;FOLD Schritt 81 = !F324 & !F328 & !E1002 & E1003 & E1004 & !E1005 & A4039  ;%{SE}%MKUKATPVW %CVW_SPS %VST_CON %P 2:Schritt 81 = !F324 & !F328 & !E1002 & E1003 & E1004 & !E1005 & A4039 , 3: ST_CON
         IF NOT $FLAG[324] AND NOT $FLAG[328] AND NOT $IN[1002] AND $IN[1003] AND $IN[1004] AND NOT $IN[1005] AND $OUT[4039] THEN
            PREVSTEP = $APP_INT[5]
            $APP_INT[5] = 81
         ENDIF
      ;ENDFOLD
   ;ENDFOLD
   ;FOLD SCHRITT 81 -- STAT EZ2/SP2/KE2-- ;%{P}%MKUKATPVW,%CSTEP,%VST_NR,%P 1:SCHRITT, 2:81, 3: STAT EZ2/SP2/KE2
      ;FOLD ;%{H}
         Case 81
      ;ENDFOLD
      ;FOLD -- Umdreh. KF setzen zwischenspeichern -- ;%{SE}%MKUKATPVW %CVW_COM %VCOMMENT %P 2:-- Umdreh. KF setzen zwischenspeichern --, 3: VW_COMMENT
      ;ENDFOLD
      ;FOLD F270 = F155 & F732 ;%{SE}%MKUKATPVW %CVW_SPS %VBOASG %P 2:F270 = F155 & F732, 3: BOASG
         $FLAG[270] = $FLAG[155] AND $FLAG[732]
      ;ENDFOLD
      ;FOLD i45 ( EIN ) = i7 ;%{SE}%MKUKATPVW %CVW_SPS %VARIASG %P 2:i45 ( EIN ) = i7, 3: ARIASG
         VW(#COUNTER,TRUE,45,$COUNT_I[7])
      ;ENDFOLD
      ;FOLD i7 ( F270 ) = i44 ;%{SE}%MKUKATPVW %CVW_SPS %VARIASG %P 2:i7 ( F270 ) = i44, 3: ARIASG
         VW(#COUNTER,$FLAG[270],7,$COUNT_I[44])
      ;ENDFOLD
      ;FOLD i1 ( EIN ) = 0 ;%{SE}%MKUKATPVW %CVW_SPS %VARIASG %P 2:i1 ( EIN ) = 0, 3: ARIASG
         VW(#COUNTER,TRUE,1,0)
      ;ENDFOLD
      ;FOLD F154 = AUS ;%{SE}%MKUKATPVW %CVW_SPS %VBOASG %P 2:F154 = AUS, 3: BOASG
         $FLAG[154] = FALSE
      ;ENDFOLD
      ;FOLD F312 = AUS ;%{SE}%MKUKATPVW %CVW_SPS %VBOASG %P 2:F312 = AUS, 3: BOASG
         $FLAG[312] = FALSE
      ;ENDFOLD
      ;FOLD F313 = AUS ;%{SE}%MKUKATPVW %CVW_SPS %VBOASG %P 2:F313 = AUS, 3: BOASG
         $FLAG[313] = FALSE
      ;ENDFOLD
      ;FOLD F324 = AUS ;%{SE}%MKUKATPVW %CVW_SPS %VBOASG %P 2:F324 = AUS, 3: BOASG
         $FLAG[324] = FALSE
      ;ENDFOLD
      ;FOLD F328 = AUS ;%{SE}%MKUKATPVW %CVW_SPS %VBOASG %P 2:F328 = AUS, 3: BOASG
         $FLAG[328] = FALSE
      ;ENDFOLD
      ;FOLD -- KF2 einschalten nach Fehler -- ;%{SE}%MKUKATPVW %CVW_COM %VCOMMENT %P 2:-- KF2 einschalten nach Fehler --, 3: VW_COMMENT
      ;ENDFOLD
      ;FOLD A994 = EIN ;%{SE}%MKUKATPVW %CVW_SPS %VBOASG %P 2:A994 = EIN, 3: BOASG
         $OUT[994] = TRUE
      ;ENDFOLD
      ;FOLD -- KF2 Versetzeinheit rueck -- ;%{SE}%MKUKATPVW %CVW_COM %VCOMMENT %P 2:-- KF2 Versetzeinheit rueck --, 3: VW_COMMENT
      ;ENDFOLD
      ;FOLD A995 = AUS ;%{SE}%MKUKATPVW %CVW_SPS %VBOASG %P 2:A995 = AUS, 3: BOASG
         $OUT[995] = FALSE
      ;ENDFOLD
      ;FOLD Schritt 82 = T11 & A4039  ;%{SE}%MKUKATPVW %CVW_SPS %VST_CON %P 2:Schritt 82 = T11 & A4039 , 3: ST_CON
         IF $TIMER_FLAG[11] AND $OUT[4039] THEN
            PREVSTEP = $APP_INT[5]
            $APP_INT[5] = 82
         ENDIF
      ;ENDFOLD
   ;ENDFOLD
   ;FOLD SCHRITT 82 -- STAT EZ2/SP2/KE2 -- ;%{P}%MKUKATPVW,%CSTEP,%VST_NR,%P 1:SCHRITT, 2:82, 3: STAT EZ2/SP2/KE2
      ;FOLD ;%{H}
         Case 82
      ;ENDFOLD
      ;FOLD F270 = AUS ;%{SE}%MKUKATPVW %CVW_SPS %VBOASG %P 2:F270 = AUS, 3: BOASG
         $FLAG[270] = FALSE
      ;ENDFOLD
      ;FOLD t11 ( EIN ) = STOP ;%{SE}%MKUKATPVW %CVW_SPS %VTSTOP %P 2:t11 ( EIN ) = STOP, 3: TSTOP
         VW(#SET_TIME,TRUE,11,1,0)
      ;ENDFOLD
      ;FOLD -- EZ2/SP2 schliessen -- ;%{SE}%MKUKATPVW %CVW_COM %VCOMMENT %P 2:-- EZ2/SP2 schliessen --, 3: VW_COMMENT
      ;ENDFOLD
      ;FOLD A877 = AUS ;%{SE}%MKUKATPVW %CVW_SPS %VBOASG %P 2:A877 = AUS, 3: BOASG
         $OUT[877] = FALSE
      ;ENDFOLD
      ;FOLD A878 = EIN ;%{SE}%MKUKATPVW %CVW_SPS %VBOASG %P 2:A878 = EIN, 3: BOASG
         $OUT[878] = TRUE
      ;ENDFOLD
      ;FOLD -- KF2 Ausblasen -- ;%{SE}%MKUKATPVW %CVW_COM %VCOMMENT %P 2:-- KF2 Ausblasen --, 3: VW_COMMENT
      ;ENDFOLD
      ;FOLD A1007 = F330 + F331 + !F330 & !F331 & !F332 ;%{SE}%MKUKATPVW %CVW_SPS %VBOASG %P 2:A1007 = F330 + F331 + !F330 & !F331 & !F332, 3: BOASG
         $OUT[1007] = $FLAG[330] OR $FLAG[331] OR NOT $FLAG[330] AND NOT $FLAG[331] AND NOT $FLAG[332]
      ;ENDFOLD
      ;FOLD Schritt 83 = (!E877 & E878 + T9) & A4039  ;%{SE}%MKUKATPVW %CVW_SPS %VST_CON %P 2:Schritt 83 = (!E877 & E878 + T9) & A4039 , 3: ST_CON
         IF (NOT $IN[877] AND $IN[878] OR $TIMER_FLAG[9]) AND $OUT[4039] THEN
            PREVSTEP = $APP_INT[5]
            $APP_INT[5] = 83
         ENDIF
      ;ENDFOLD
   ;ENDFOLD
   ;FOLD SCHRITT 83 -- STAT EZ2/SP2/KE2 -- ;%{P}%MKUKATPVW,%CSTEP,%VST_NR,%P 1:SCHRITT, 2:83, 3: STAT EZ2/SP2/KE2
      ;FOLD ;%{H}
         Case 83
      ;ENDFOLD
      ;FOLD -- RSK Fehlerausgabe Kraftaufbau -- ;%{SE}%MKUKATPVW %CVW_COM %VCOMMENT %P 2:-- RSK Fehlerausgabe Kraftaufbau --, 3: VW_COMMENT
      ;ENDFOLD
      ;FOLD F325 = T9 ;%{SE}%MKUKATPVW %CVW_SPS %VBOASG %P 2:F325 = T9, 3: BOASG
         $FLAG[325] = $TIMER_FLAG[9]
      ;ENDFOLD
      ;FOLD -- RSK Sammelstoerung -- ;%{SE}%MKUKATPVW %CVW_COM %VCOMMENT %P 2:-- RSK Sammelstoerung --, 3: VW_COMMENT
      ;ENDFOLD
      ;FOLD F329 = F325 ;%{SE}%MKUKATPVW %CVW_SPS %VBOASG %P 2:F329 = F325, 3: BOASG
         $FLAG[329] = $FLAG[325]
      ;ENDFOLD
      ;FOLD -- KF2 abschalten bei Fehler -- ;%{SE}%MKUKATPVW %CVW_COM %VCOMMENT %P 2:-- KF2 abschalten bei Fehler --, 3: VW_COMMENT
      ;ENDFOLD
      ;FOLD A994 = !T9 ;%{SE}%MKUKATPVW %CVW_SPS %VBOASG %P 2:A994 = !T9, 3: BOASG
         $OUT[994] = NOT $TIMER_FLAG[9]
      ;ENDFOLD
      ;FOLD -- KF2 Ausblasen -- ;%{SE}%MKUKATPVW %CVW_COM %VCOMMENT %P 2:-- KF2 Ausblasen --, 3: VW_COMMENT
      ;ENDFOLD
      ;FOLD A1007 = (F330 + F331 + !F330 & !F331 & !F332) & !T9 ;%{SE}%MKUKATPVW %CVW_SPS %VBOASG %P 2:A1007 = (F330 + F331 + !F330 & !F331 & !F332) & !T9, 3: BOASG
         $OUT[1007] = ($FLAG[330] OR $FLAG[331] OR NOT $FLAG[330] AND NOT $FLAG[331] AND NOT $FLAG[332]) AND NOT $TIMER_FLAG[9]
      ;ENDFOLD
      ;FOLD -- Warte Fraesen fertig oder Timeout -- ;%{SE}%MKUKATPVW %CVW_COM %VCOMMENT %P 2:-- Warte Fraesen fertig oder Timeout --, 3: VW_COMMENT
      ;ENDFOLD
      ;FOLD Schritt 84 = (F139 & F154 + F138 & F150 & !F287 + T7 + T9 + F325) & A4039  ;%{SE}%MKUKATPVW %CVW_SPS %VST_CON %P 2:Schritt 84 = (F139 & F154 + F138 & F150 & !F287 + T7 + T9 + F325) & A4039 , 3: ST_CON
         IF ($FLAG[139] AND $FLAG[154] OR $FLAG[138] AND $FLAG[150] AND NOT $FLAG[287] OR $TIMER_FLAG[7] OR $TIMER_FLAG[9] OR $FLAG[325]) AND $OUT[4039] THEN
            PREVSTEP = $APP_INT[5]
            $APP_INT[5] = 84
         ENDIF
      ;ENDFOLD
      ;FOLD Schritt 84 = (F138 & F152 & F287 + T7 + T9 + F325) & A4039  ;%{SE}%MKUKATPVW %CVW_SPS %VST_CON %P 2:Schritt 84 = (F138 & F152 & F287 + T7 + T9 + F325) & A4039 , 3: ST_CON
         IF ($FLAG[138] AND $FLAG[152] AND $FLAG[287] OR $TIMER_FLAG[7] OR $TIMER_FLAG[9] OR $FLAG[325]) AND $OUT[4039] THEN
            PREVSTEP = $APP_INT[5]
            $APP_INT[5] = 84
         ENDIF
      ;ENDFOLD
   ;ENDFOLD
   ;FOLD SCHRITT 84 -- STAT EZ2/SP2/KE2-- ;%{P}%MKUKATPVW,%CSTEP,%VST_NR,%P 1:SCHRITT, 2:84, 3: STAT EZ2/SP2/KE2
      ;FOLD ;%{H}
         Case 84
      ;ENDFOLD
      ;FOLD t9 ( EIN ) = STOP ;%{SE}%MKUKATPVW %CVW_SPS %VTSTOP %P 2:t9 ( EIN ) = STOP, 3: TSTOP
         VW(#SET_TIME,TRUE,9,1,0)
      ;ENDFOLD
      ;FOLD -- EZ2/SP2/KE2 oeffnen -- ;%{SE}%MKUKATPVW %CVW_COM %VCOMMENT %P 2:-- EZ2/SP2/KE2 oeffnen --, 3: VW_COMMENT
      ;ENDFOLD
      ;FOLD A878 = AUS ;%{SE}%MKUKATPVW %CVW_SPS %VBOASG %P 2:A878 = AUS, 3: BOASG
         $OUT[878] = FALSE
      ;ENDFOLD
      ;FOLD A877 = EIN ;%{SE}%MKUKATPVW %CVW_SPS %VBOASG %P 2:A877 = EIN, 3: BOASG
         $OUT[877] = TRUE
      ;ENDFOLD
      ;FOLD -- KF2 Ausblasen -- ;%{SE}%MKUKATPVW %CVW_COM %VCOMMENT %P 2:-- KF2 Ausblasen --, 3: VW_COMMENT
      ;ENDFOLD
      ;FOLD A1007 = F330 + F331 + F332 + !F330 & !F331 & !F332 ;%{SE}%MKUKATPVW %CVW_SPS %VBOASG %P 2:A1007 = F330 + F331 + F332 + !F330 & !F331 & !F332, 3: BOASG
         $OUT[1007] = $FLAG[330] OR $FLAG[331] OR $FLAG[332] OR NOT $FLAG[330] AND NOT $FLAG[331] AND NOT $FLAG[332]
      ;ENDFOLD
      ;FOLD -- KF Ausblasen Ausschaltverzoegerung starten -- ;%{SE}%MKUKATPVW %CVW_COM %VCOMMENT %P 2:-- KF Ausblasen Ausschaltverzoegerung starten --, 3: VW_COMMENT
      ;ENDFOLD
      ;FOLD F738 = EIN ;%{SE}%MKUKATPVW %CVW_SPS %VBOASG %P 2:F738 = EIN, 3: BOASG
         $FLAG[738] = TRUE
      ;ENDFOLD
      ;FOLD -- RSK Sammelstoerung -- ;%{SE}%MKUKATPVW %CVW_COM %VCOMMENT %P 2:-- RSK Sammelstoerung --, 3: VW_COMMENT
      ;ENDFOLD
      ;FOLD F329 = T7 + T9 + F325 ;%{SE}%MKUKATPVW %CVW_SPS %VBOASG %P 2:F329 = T7 + T9 + F325, 3: BOASG
         $FLAG[329] = $TIMER_FLAG[7] OR $TIMER_FLAG[9] OR $FLAG[325]
      ;ENDFOLD
      ;FOLD -- Hilfsflag Startfraesen -- ;%{SE}%MKUKATPVW %CVW_COM %VCOMMENT %P 2:-- Hilfsflag Startfraesen --, 3: VW_COMMENT
      ;ENDFOLD
      ;FOLD F152 = (F152 & F138 + F154 & F139) & F287 ;%{SE}%MKUKATPVW %CVW_SPS %VBOASG %P 2:F152 = (F152 & F138 + F154 & F139) & F287, 3: BOASG
         $FLAG[152] = ($FLAG[152] AND $FLAG[138] OR $FLAG[154] AND $FLAG[139]) AND $FLAG[287]
      ;ENDFOLD
      ;FOLD F154 = !F164 & F154 + F164 & F287 & F154 ;%{SE}%MKUKATPVW %CVW_SPS %VBOASG %P 2:F154 = !F164 & F154 + F164 & F287 & F154, 3: BOASG
         $FLAG[154] = NOT $FLAG[164] AND $FLAG[154] OR $FLAG[164] AND $FLAG[287] AND $FLAG[154]
      ;ENDFOLD
      ;FOLD F287 = F138 + F139 & F164 ;%{SE}%MKUKATPVW %CVW_SPS %VBOASG %P 2:F287 = F138 + F139 & F164, 3: BOASG
         $FLAG[287] = $FLAG[138] OR $FLAG[139] AND $FLAG[164]
      ;ENDFOLD
      ;FOLD -- Neues Fraesprogramm und Zaehler ruecksetzen -- ;%{SE}%MKUKATPVW %CVW_COM %VCOMMENT %P 2:-- Neues Fraesprogramm und Zaehler ruecksetzen --, 3: VW_COMMENT
      ;ENDFOLD
      ;FOLD F270 = F152 & F732 ;%{SE}%MKUKATPVW %CVW_SPS %VBOASG %P 2:F270 = F152 & F732, 3: BOASG
         $FLAG[270] = $FLAG[152] AND $FLAG[732]
      ;ENDFOLD
      ;FOLD bin6 ( F732 ) = 36 ;%{SE}%MKUKATPVW %CVW_SPS %VARIASG %P 2:bin6 ( F732 ) = 36, 3: ARIASG
         VW(#BINOUT,$FLAG[732],6,36)
      ;ENDFOLD
      ;FOLD i7 ( F270 ) = i45 ;%{SE}%MKUKATPVW %CVW_SPS %VARIASG %P 2:i7 ( F270 ) = i45, 3: ARIASG
         VW(#COUNTER,$FLAG[270],7,$COUNT_I[45])
      ;ENDFOLD
      ;FOLD -- Wiederholung beim Startfraesen -- ;%{SE}%MKUKATPVW %CVW_COM %VCOMMENT %P 2:-- Wiederholung beim Startfraesen --, 3: VW_COMMENT
      ;ENDFOLD
      ;FOLD Schritt 81 = E877 & !E878 & (F138 & !F152 + F139 & F164 & !F152) & !F325 & !F329 & A4039  ;%{SE}%MKUKATPVW %CVW_SPS %VST_CON %P 2:Schritt 81 = E877 & !E878 & (F138 & !F152 + F139 & F164 & !F152) & !F325 & !F329 & A4039 , 3: ST_CON
         IF $IN[877] AND NOT $IN[878] AND ($FLAG[138] AND NOT $FLAG[152] OR $FLAG[139] AND $FLAG[164] AND NOT $FLAG[152]) AND NOT $FLAG[325] AND NOT $FLAG[329] AND $OUT[4039] THEN
            PREVSTEP = $APP_INT[5]
            $APP_INT[5] = 81
         ENDIF
      ;ENDFOLD
      ;FOLD -- Weiter wenn Fraesen fertig -- ;%{SE}%MKUKATPVW %CVW_COM %VCOMMENT %P 2:-- Weiter wenn Fraesen fertig --, 3: VW_COMMENT
      ;ENDFOLD
      ;FOLD Schritt 85 = E877 & !E878 & (F139 & F154 & (!F164 + F152) + F138 & F152 + F325 + F329) & A4039  ;%{SE}%MKUKATPVW %CVW_SPS %VST_CON %P 2:Schritt 85 = E877 & !E878 & (F139 & F154 & (!F164 + F152) + F138 & F152 + F325 + F329) & A4039 , 3: ST_CON
         IF $IN[877] AND NOT $IN[878] AND ($FLAG[139] AND $FLAG[154] AND (NOT $FLAG[164] OR $FLAG[152]) OR $FLAG[138] AND $FLAG[152] OR $FLAG[325] OR $FLAG[329]) AND $OUT[4039] THEN
            PREVSTEP = $APP_INT[5]
            $APP_INT[5] = 85
         ENDIF
      ;ENDFOLD
   ;ENDFOLD
   ;FOLD SCHRITT 85 -- STAT EZ2/SP2/KE2-- ;%{P}%MKUKATPVW,%CSTEP,%VST_NR,%P 1:SCHRITT, 2:85, 3: STAT EZ2/SP2/KE2
      ;FOLD ;%{H}
         Case 85
      ;ENDFOLD
      ;FOLD F324 = AUS ;%{SE}%MKUKATPVW %CVW_SPS %VBOASG %P 2:F324 = AUS, 3: BOASG
         $FLAG[324] = FALSE
      ;ENDFOLD
      ;FOLD A877 = AUS ;%{SE}%MKUKATPVW %CVW_SPS %VBOASG %P 2:A877 = AUS, 3: BOASG
         $OUT[877] = FALSE
      ;ENDFOLD
      ;FOLD -- KF2 abschalten -- ;%{SE}%MKUKATPVW %CVW_COM %VCOMMENT %P 2:-- KF2 abschalten --, 3: VW_COMMENT
      ;ENDFOLD
      ;FOLD A994 = AUS ;%{SE}%MKUKATPVW %CVW_SPS %VBOASG %P 2:A994 = AUS, 3: BOASG
         $OUT[994] = FALSE
      ;ENDFOLD
      ;FOLD -- Ueberwachungszeit KF2 Versetzeinheit -- ;%{SE}%MKUKATPVW %CVW_COM %VCOMMENT %P 2:-- Ueberwachungszeit KF2 Versetzeinheit --, 3: VW_COMMENT
      ;ENDFOLD
      ;FOLD t8 ( EIN ) = -40[1/10Sek] ;%{SE}%MKUKATPVW %CVW_SPS %VTASG %P 2:t8 ( EIN ) = -40[1/10Sek], 3: TASG
         VW(#SET_TIME,TRUE,8,0,-40)
      ;ENDFOLD
      ;FOLD Schritt 86 = A4039  ;%{SE}%MKUKATPVW %CVW_SPS %VST_CON %P 2:Schritt 86 = A4039 , 3: ST_CON
         IF $OUT[4039] THEN
            PREVSTEP = $APP_INT[5]
            $APP_INT[5] = 86
         ENDIF
      ;ENDFOLD
   ;ENDFOLD
   ;FOLD SCHRITT 86 -- STAT EZ2/SP2/KE2 -- ;%{P}%MKUKATPVW,%CSTEP,%VST_NR,%P 1:SCHRITT, 2:86, 3: STAT EZ2/SP2/KE2
      ;FOLD ;%{H}
         Case 86
      ;ENDFOLD
      ;FOLD F328 = AUS ;%{SE}%MKUKATPVW %CVW_SPS %VBOASG %P 2:F328 = AUS, 3: BOASG
         $FLAG[328] = FALSE
      ;ENDFOLD
      ;FOLD -- KF2 Versetzeinheit vor -- ;%{SE}%MKUKATPVW %CVW_COM %VCOMMENT %P 2:-- KF2 Versetzeinheit vor --, 3: VW_COMMENT
      ;ENDFOLD
      ;FOLD A995 = F564 ;%{SE}%MKUKATPVW %CVW_SPS %VBOASG %P 2:A995 = F564, 3: BOASG
         $OUT[995] = $FLAG[564]
      ;ENDFOLD
      ;FOLD -- RSK Fehlerausgabe KS2 Arbeitsst. -- ;%{SE}%MKUKATPVW %CVW_COM %VCOMMENT %P 2:-- RSK Fehlerausgabe KS2 Arbeitsst. --, 3: VW_COMMENT
      ;ENDFOLD
      ;FOLD F324 = (E1002 + !E1003 + !E1004 + E1005) & !F323 & !F328 + F324 ;%{SE}%MKUKATPVW %CVW_SPS %VBOASG %P 2:F324 = (E1002 + !E1003 + !E1004 + E1005) & !F323 & !F328 + F324, 3: BOASG
         $FLAG[324] = ($IN[1002] OR NOT $IN[1003] OR NOT $IN[1004] OR $IN[1005]) AND NOT $FLAG[323] AND NOT $FLAG[328] OR $FLAG[324]
      ;ENDFOLD
      ;FOLD -- RSK Sammelstoerung -- ;%{SE}%MKUKATPVW %CVW_COM %VCOMMENT %P 2:-- RSK Sammelstoerung --, 3: VW_COMMENT
      ;ENDFOLD
      ;FOLD F329 = F324 + F325 ;%{SE}%MKUKATPVW %CVW_SPS %VBOASG %P 2:F329 = F324 + F325, 3: BOASG
         $FLAG[329] = $FLAG[324] OR $FLAG[325]
      ;ENDFOLD
      ;FOLD -- Ueberwachungszeit KS2 schwenken -- ;%{SE}%MKUKATPVW %CVW_COM %VCOMMENT %P 2:-- Ueberwachungszeit KS2 schwenken --, 3: VW_COMMENT
      ;ENDFOLD
      ;FOLD t9 ( EIN ) = -100[1/10Sek] ;%{SE}%MKUKATPVW %CVW_SPS %VTASG %P 2:t9 ( EIN ) = -100[1/10Sek], 3: TASG
         VW(#SET_TIME,TRUE,9,0,-100)
      ;ENDFOLD
      ;FOLD Schritt 85 = F324 & (E26 + E27) & A4039  ;%{SE}%MKUKATPVW %CVW_SPS %VST_CON %P 2:Schritt 85 = F324 & (E26 + E27) & A4039 , 3: ST_CON
         IF $FLAG[324] AND ($IN[26] OR $IN[27]) AND $OUT[4039] THEN
            PREVSTEP = $APP_INT[5]
            $APP_INT[5] = 85
         ENDIF
      ;ENDFOLD
      ;FOLD Schritt 87 = (!F324 & (E995 & F564 + !E995 & !F564) + T8 + F325) & A4039  ;%{SE}%MKUKATPVW %CVW_SPS %VST_CON %P 2:Schritt 87 = (!F324 & (E995 & F564 + !E995 & !F564) + T8 + F325) & A4039 , 3: ST_CON
         IF (NOT $FLAG[324] AND ($IN[995] AND $FLAG[564] OR NOT $IN[995] AND NOT $FLAG[564]) OR $TIMER_FLAG[8] OR $FLAG[325]) AND $OUT[4039] THEN
            PREVSTEP = $APP_INT[5]
            $APP_INT[5] = 87
         ENDIF
      ;ENDFOLD
   ;ENDFOLD
   ;FOLD SCHRITT 87 -- STAT EZ2/SP2/KE2-- ;%{P}%MKUKATPVW,%CSTEP,%VST_NR,%P 1:SCHRITT, 2:87, 3: STAT EZ2/SP2/KE2
      ;FOLD ;%{H}
         Case 87
      ;ENDFOLD
      ;FOLD F323 = AUS ;%{SE}%MKUKATPVW %CVW_SPS %VBOASG %P 2:F323 = AUS, 3: BOASG
         $FLAG[323] = FALSE
      ;ENDFOLD
      ;FOLD F328 = AUS ;%{SE}%MKUKATPVW %CVW_SPS %VBOASG %P 2:F328 = AUS, 3: BOASG
         $FLAG[328] = FALSE
      ;ENDFOLD
      ;FOLD -- RSK Sammelstoerung -- ;%{SE}%MKUKATPVW %CVW_COM %VCOMMENT %P 2:-- RSK Sammelstoerung --, 3: VW_COMMENT
      ;ENDFOLD
      ;FOLD F329 = F325 ;%{SE}%MKUKATPVW %CVW_SPS %VBOASG %P 2:F329 = F325, 3: BOASG
         $FLAG[329] = $FLAG[325]
      ;ENDFOLD
      ;FOLD -- KF2 ein -- ;%{SE}%MKUKATPVW %CVW_COM %VCOMMENT %P 2:-- KF2 ein --, 3: VW_COMMENT
      ;ENDFOLD
      ;FOLD A994 = EIN ;%{SE}%MKUKATPVW %CVW_SPS %VBOASG %P 2:A994 = EIN, 3: BOASG
         $OUT[994] = TRUE
      ;ENDFOLD
      ;FOLD -- KS2 in Ruhestellung schwenken -- ;%{SE}%MKUKATPVW %CVW_COM %VCOMMENT %P 2:-- KS2 in Ruhestellung schwenken --, 3: VW_COMMENT
      ;ENDFOLD
      ;FOLD A1002 = (F746 + !F714) & (E877 + F714) & (E995 & F564 + !E995 & !F564) ;%{SE}%MKUKATPVW %CVW_SPS %VBOASG %P 2:A1002 = (F746 + !F714) & (E877 + F714) & (E995 & F564 + !E995 & !F564), 3: BOASG
         $OUT[1002] = ($FLAG[746] OR NOT $FLAG[714]) AND ($IN[877] OR $FLAG[714]) AND ($IN[995] AND $FLAG[564] OR NOT $IN[995] AND NOT $FLAG[564])
      ;ENDFOLD
      ;FOLD Schritt 88 = (F746 + !F714 + T9) & (A1002 + T9) & (E877 + F714) & A4039  ;%{SE}%MKUKATPVW %CVW_SPS %VST_CON %P 2:Schritt 88 = (F746 + !F714 + T9) & (A1002 + T9) & (E877 + F714) & A4039 , 3: ST_CON
         IF ($FLAG[746] OR NOT $FLAG[714] OR $TIMER_FLAG[9]) AND ($OUT[1002] OR $TIMER_FLAG[9]) AND ($IN[877] OR $FLAG[714]) AND $OUT[4039] THEN
            PREVSTEP = $APP_INT[5]
            $APP_INT[5] = 88
         ENDIF
      ;ENDFOLD
   ;ENDFOLD
   ;FOLD SCHRITT 88 -- STAT EZ2/SP2 -- ;%{P}%MKUKATPVW,%CSTEP,%VST_NR,%P 1:SCHRITT, 2:88, 3: STAT EZ2/SP2
      ;FOLD ;%{H}
         Case 88
      ;ENDFOLD
      ;FOLD -- Hilfsflag SK Programmwechsel -- ;%{SE}%MKUKATPVW %CVW_COM %VCOMMENT %P 2:-- Hilfsflag SK Programmwechsel --, 3: VW_COMMENT
      ;ENDFOLD
      ;FOLD F334 = AUS ;%{SE}%MKUKATPVW %CVW_SPS %VBOASG %P 2:F334 = AUS, 3: BOASG
         $FLAG[334] = FALSE
      ;ENDFOLD
      ;FOLD -- RSK Fehlerausgabe KF Versetzeinheit -- ;%{SE}%MKUKATPVW %CVW_COM %VCOMMENT %P 2:-- RSK Fehlerausgabe KF Versetzeinheit --, 3: VW_COMMENT
      ;ENDFOLD
      ;FOLD F328 = !E995 & F564 & !F323 + F328 ;%{SE}%MKUKATPVW %CVW_SPS %VBOASG %P 2:F328 = !E995 & F564 & !F323 + F328, 3: BOASG
         $FLAG[328] = NOT $IN[995] AND $FLAG[564] AND NOT $FLAG[323] OR $FLAG[328]
      ;ENDFOLD
      ;FOLD -- RSK Fehlerausgabe KS2 Ruhestellung -- ;%{SE}%MKUKATPVW %CVW_COM %VCOMMENT %P 2:-- RSK Fehlerausgabe KS2 Ruhestellung --, 3: VW_COMMENT
      ;ENDFOLD
      ;FOLD F323 = (!E1002 + E1003 + E1004 + !E1005) & T9 & (E995 + !F564) + F323 ;%{SE}%MKUKATPVW %CVW_SPS %VBOASG %P 2:F323 = (!E1002 + E1003 + E1004 + !E1005) & T9 & (E995 + !F564) + F323, 3: BOASG
         $FLAG[323] = (NOT $IN[1002] OR $IN[1003] OR $IN[1004] OR NOT $IN[1005]) AND $TIMER_FLAG[9] AND ($IN[995] OR NOT $FLAG[564]) OR $FLAG[323]
      ;ENDFOLD
      ;FOLD -- RSK Fehlerausgabe EZ/SP min. Oeffnung -- ;%{SE}%MKUKATPVW %CVW_COM %VCOMMENT %P 2:-- RSK Fehlerausgabe EZ/SP min. Oeffnung --, 3: VW_COMMENT
      ;ENDFOLD
      ;FOLD F333 = !F746 ;%{SE}%MKUKATPVW %CVW_SPS %VBOASG %P 2:F333 = !F746, 3: BOASG
         $FLAG[333] = NOT $FLAG[746]
      ;ENDFOLD
      ;FOLD -- RSK Sammelstoerung -- ;%{SE}%MKUKATPVW %CVW_COM %VCOMMENT %P 2:-- RSK Sammelstoerung --, 3: VW_COMMENT
      ;ENDFOLD
      ;FOLD F329 = F323 + F325 + F328 + F333 ;%{SE}%MKUKATPVW %CVW_SPS %VBOASG %P 2:F329 = F323 + F325 + F328 + F333, 3: BOASG
         $FLAG[329] = $FLAG[323] OR $FLAG[325] OR $FLAG[328] OR $FLAG[333]
      ;ENDFOLD
      ;FOLD A994 = !F323 & !F328 ;%{SE}%MKUKATPVW %CVW_SPS %VBOASG %P 2:A994 = !F323 & !F328, 3: BOASG
         $OUT[994] = NOT $FLAG[323] AND NOT $FLAG[328]
      ;ENDFOLD
      ;FOLD A995 = F564 ;%{SE}%MKUKATPVW %CVW_SPS %VBOASG %P 2:A995 = F564, 3: BOASG
         $OUT[995] = $FLAG[564]
      ;ENDFOLD
      ;FOLD Schritt 86 = (F323 + F328) & (E26 + E27) & A4039  ;%{SE}%MKUKATPVW %CVW_SPS %VST_CON %P 2:Schritt 86 = (F323 + F328) & (E26 + E27) & A4039 , 3: ST_CON
         IF ($FLAG[323] OR $FLAG[328]) AND ($IN[26] OR $IN[27]) AND $OUT[4039] THEN
            PREVSTEP = $APP_INT[5]
            $APP_INT[5] = 86
         ENDIF
      ;ENDFOLD
      ;FOLD Schritt 89 = !A1002 & E1002 & !E1003 & !E1004 & E1005 & A4039  ;%{SE}%MKUKATPVW %CVW_SPS %VST_CON %P 2:Schritt 89 = !A1002 & E1002 & !E1003 & !E1004 & E1005 & A4039 , 3: ST_CON
         IF NOT $OUT[1002] AND $IN[1002] AND NOT $IN[1003] AND NOT $IN[1004] AND $IN[1005] AND $OUT[4039] THEN
            PREVSTEP = $APP_INT[5]
            $APP_INT[5] = 89
         ENDIF
      ;ENDFOLD
   ;ENDFOLD
   ;FOLD SCHRITT 89 -- STAT EZ2/SP2/KE2 -- ;%{P}%MKUKATPVW,%CSTEP,%VST_NR,%P 1:SCHRITT, 2:89, 3: STAT EZ2/SP2/KE2
      ;FOLD ;%{H}
         Case 89
      ;ENDFOLD
      ;FOLD F323 = AUS ;%{SE}%MKUKATPVW %CVW_SPS %VBOASG %P 2:F323 = AUS, 3: BOASG
         $FLAG[323] = FALSE
      ;ENDFOLD
      ;FOLD F328 = AUS ;%{SE}%MKUKATPVW %CVW_SPS %VBOASG %P 2:F328 = AUS, 3: BOASG
         $FLAG[328] = FALSE
      ;ENDFOLD
      ;FOLD -- RSK Sammelstoerung -- ;%{SE}%MKUKATPVW %CVW_COM %VCOMMENT %P 2:-- RSK Sammelstoerung --, 3: VW_COMMENT
      ;ENDFOLD
      ;FOLD F329 = F325 ;%{SE}%MKUKATPVW %CVW_SPS %VBOASG %P 2:F329 = F325, 3: BOASG
         $FLAG[329] = $FLAG[325]
      ;ENDFOLD
      ;FOLD t9 ( EIN ) = STOP ;%{SE}%MKUKATPVW %CVW_SPS %VTSTOP %P 2:t9 ( EIN ) = STOP, 3: TSTOP
         VW(#SET_TIME,TRUE,9,1,0)
      ;ENDFOLD
      ;FOLD -- KF2 Versetzeinheit rueck -- ;%{SE}%MKUKATPVW %CVW_COM %VCOMMENT %P 2:-- KF2 Versetzeinheit rueck --, 3: VW_COMMENT
      ;ENDFOLD
      ;FOLD A995 = AUS ;%{SE}%MKUKATPVW %CVW_SPS %VBOASG %P 2:A995 = AUS, 3: BOASG
         $OUT[995] = FALSE
      ;ENDFOLD
      ;FOLD -- KF2 aus -- ;%{SE}%MKUKATPVW %CVW_COM %VCOMMENT %P 2:-- KF2 aus --, 3: VW_COMMENT
      ;ENDFOLD
      ;FOLD A994 = AUS ;%{SE}%MKUKATPVW %CVW_SPS %VBOASG %P 2:A994 = AUS, 3: BOASG
         $OUT[994] = FALSE
      ;ENDFOLD
      ;FOLD -- KF1 Ausblasen -- ;%{SE}%MKUKATPVW %CVW_COM %VCOMMENT %P 2:-- KF1 Ausblasen --, 3: VW_COMMENT
      ;ENDFOLD
      ;FOLD A1007 = (F330 + F331 + F332) & F738 ;%{SE}%MKUKATPVW %CVW_SPS %VBOASG %P 2:A1007 = (F330 + F331 + F332) & F738, 3: BOASG
         $OUT[1007] = ($FLAG[330] OR $FLAG[331] OR $FLAG[332]) AND $FLAG[738]
      ;ENDFOLD
      ;FOLD bin3 ( F285 ) = 5 ;%{SE}%MKUKATPVW %CVW_SPS %VARIASG %P 2:bin3 ( F285 ) = 5, 3: ARIASG
         VW(#BINOUT,$FLAG[285],3,5)
      ;ENDFOLD
      ;FOLD bin6 ( !F285 ) = 1 ;%{SE}%MKUKATPVW %CVW_SPS %VARIASG %P 2:bin6 ( !F285 ) = 1, 3: ARIASG
         VW(#BINOUT,NOT $FLAG[285],6,1)
      ;ENDFOLD
      ;FOLD -- Wartezeit Programmwechsel SK -- ;%{SE}%MKUKATPVW %CVW_COM %VCOMMENT %P 2:-- Wartezeit Programmwechsel SK --, 3: VW_COMMENT
      ;ENDFOLD
      ;FOLD T8 ( !F334 ) = -2[1/10Sek] ;%{SE}%MKUKATPVW %CVW_SPS %VTASG %P 2:T8 ( !F334 ) = -2[1/10Sek], 3: TASG
         VW(#SET_TIME,NOT $FLAG[334],8,0,-2)
      ;ENDFOLD
      ;FOLD -- Hilfsflag SK Programmwechsel -- ;%{SE}%MKUKATPVW %CVW_COM %VCOMMENT %P 2:-- Hilfsflag SK Programmwechsel --, 3: VW_COMMENT
      ;ENDFOLD
      ;FOLD F334 = EIN ;%{SE}%MKUKATPVW %CVW_SPS %VBOASG %P 2:F334 = EIN, 3: BOASG
         $FLAG[334] = TRUE
      ;ENDFOLD
      ;FOLD -- Ueberwachungszeit EZ2/SP2/KE2 Messen -- ;%{SE}%MKUKATPVW %CVW_COM %VCOMMENT %P 2:-- Ueberwachungszeit EZ2/SP2/KE2 Messen --, 3: VW_COMMENT
      ;ENDFOLD
      ;FOLD t9 ( EIN ) = -150[1/10Sek] ;%{SE}%MKUKATPVW %CVW_SPS %VTASG %P 2:t9 ( EIN ) = -150[1/10Sek], 3: TASG
         VW(#SET_TIME,TRUE,9,0,-150)
      ;ENDFOLD
      ;FOLD Schritt 74 = (F325 + F329) & (E26 + E27) & A4039  ;%{SE}%MKUKATPVW %CVW_SPS %VST_CON %P 2:Schritt 74 = (F325 + F329) & (E26 + E27) & A4039 , 3: ST_CON
         IF ($FLAG[325] OR $FLAG[329]) AND ($IN[26] OR $IN[27]) AND $OUT[4039] THEN
            PREVSTEP = $APP_INT[5]
            $APP_INT[5] = 74
         ENDIF
      ;ENDFOLD
      ;FOLD Schritt 90 = T8 & !F325 & !F329 & A4039  ;%{SE}%MKUKATPVW %CVW_SPS %VST_CON %P 2:Schritt 90 = T8 & !F325 & !F329 & A4039 , 3: ST_CON
         IF $TIMER_FLAG[8] AND NOT $FLAG[325] AND NOT $FLAG[329] AND $OUT[4039] THEN
            PREVSTEP = $APP_INT[5]
            $APP_INT[5] = 90
         ENDIF
      ;ENDFOLD
   ;ENDFOLD
   ;FOLD SCHRITT 90 -- STAT EZ2/SP2/KE2 -- ;%{P}%MKUKATPVW,%CSTEP,%VST_NR,%P 1:SCHRITT, 2:90, 3: STAT EZ2/SP2/KE2
      ;FOLD ;%{H}
         Case 90
      ;ENDFOLD
      ;FOLD -- Hilfsflag SK Programmwechsel -- ;%{SE}%MKUKATPVW %CVW_COM %VCOMMENT %P 2:-- Hilfsflag SK Programmwechsel --, 3: VW_COMMENT
      ;ENDFOLD
      ;FOLD F334 = AUS ;%{SE}%MKUKATPVW %CVW_SPS %VBOASG %P 2:F334 = AUS, 3: BOASG
         $FLAG[334] = FALSE
      ;ENDFOLD
      ;FOLD -- Quitt. Fraesen SK2/SK1 -- ;%{SE}%MKUKATPVW %CVW_COM %VCOMMENT %P 2:-- Quitt. Fraesen SK2/SK1 --, 3: VW_COMMENT
      ;ENDFOLD
      ;FOLD A946 = (!F285 & !F329 & !F322 & !F831) + (F831 & A946) ;%{SE}%MKUKATPVW %CVW_SPS %VBOASG %P 2:A946 = (!F285 & !F329 & !F322 & !F831) + (F831 & A946), 3: BOASG
         $OUT[946] = (NOT $FLAG[285] AND NOT $FLAG[329] AND NOT $FLAG[322] AND NOT $FLAG[831]) OR ($FLAG[831] AND $OUT[946])
      ;ENDFOLD
      ;FOLD A786 = (F285 & !F329 & !F322 & !F831 & !F830) + (F830 & A786) ;%{SE}%MKUKATPVW %CVW_SPS %VBOASG %P 2:A786 = (F285 & !F329 & !F322 & !F831 & !F830) + (F830 & A786), 3: BOASG
         $OUT[786] = ($FLAG[285] AND NOT $FLAG[329] AND NOT $FLAG[322] AND NOT $FLAG[831] AND NOT $FLAG[830]) OR ($FLAG[830] AND $OUT[786])
      ;ENDFOLD
      ;FOLD A882 = (!F285 & !F329 & !F322 & F831) + (!F831 & A882) ;%{SE}%MKUKATPVW %CVW_SPS %VBOASG %P 2:A882 = (!F285 & !F329 & !F322 & F831) + (!F831 & A882), 3: BOASG
         $OUT[882] = (NOT $FLAG[285] AND NOT $FLAG[329] AND NOT $FLAG[322] AND $FLAG[831]) OR (NOT $FLAG[831] AND $OUT[882])
      ;ENDFOLD
      ;FOLD -- RSK Sammelstoerung -- ;%{SE}%MKUKATPVW %CVW_COM %VCOMMENT %P 2:-- RSK Sammelstoerung --, 3: VW_COMMENT
      ;ENDFOLD
      ;FOLD F329 = T9 ;%{SE}%MKUKATPVW %CVW_SPS %VBOASG %P 2:F329 = T9, 3: BOASG
         $FLAG[329] = $TIMER_FLAG[9]
      ;ENDFOLD
      ;FOLD -- Messen nach Fraesen -- ;%{SE}%MKUKATPVW %CVW_COM %VCOMMENT %P 2:-- Messen nach Fraesen --, 3: VW_COMMENT
      ;ENDFOLD
      ;FOLD A919 = (!F138 & F139 & !F831) + (F831 & A919) ;%{SE}%MKUKATPVW %CVW_SPS %VBOASG %P 2:A919 = (!F138 & F139 & !F831) + (F831 & A919), 3: BOASG
         $OUT[919] = (NOT $FLAG[138] AND $FLAG[139] AND NOT $FLAG[831]) OR ($FLAG[831] AND $OUT[919])
      ;ENDFOLD
      ;FOLD A918 = (F138 & !F139 & !F831) + (F831 & A918) ;%{SE}%MKUKATPVW %CVW_SPS %VBOASG %P 2:A918 = (F138 & !F139 & !F831) + (F831 & A918), 3: BOASG
         $OUT[918] = ($FLAG[138] AND NOT $FLAG[139] AND NOT $FLAG[831]) OR ($FLAG[831] AND $OUT[918])
      ;ENDFOLD
      ;FOLD F836 = (F138 + F139) & !F329 ;%{SE}%MKUKATPVW %CVW_SPS %VBOASG %P 2:F836 = (F138 + F139) & !F329, 3: BOASG
         $FLAG[836] = ($FLAG[138] OR $FLAG[139]) AND NOT $FLAG[329]
      ;ENDFOLD
      ;FOLD A917 = (F836 & !F831) + (F831 & A917) ;%{SE}%MKUKATPVW %CVW_SPS %VBOASG %P 2:A917 = (F836 & !F831) + (F831 & A917), 3: BOASG
         $OUT[917] = ($FLAG[836] AND NOT $FLAG[831]) OR ($FLAG[831] AND $OUT[917])
      ;ENDFOLD
      ;FOLD A885 = (F836 & F831) + (!F831 & A885) ;%{SE}%MKUKATPVW %CVW_SPS %VBOASG %P 2:A885 = (F836 & F831) + (!F831 & A885), 3: BOASG
         $OUT[885] = ($FLAG[836] AND $FLAG[831]) OR (NOT $FLAG[831] AND $OUT[885])
      ;ENDFOLD
      ;FOLD F836 = (!E882 & E884 & !E883) & F831 & A4039 ;%{SE}%MKUKATPVW %CVW_SPS %VBOASG %P 2:F836 = (!E882 & E884 & !E883) & F831 & A4039, 3: BOASG
         $FLAG[836] = (NOT $IN[882] AND $IN[884] AND NOT $IN[883]) AND $FLAG[831] AND $OUT[4039]
      ;ENDFOLD
      ;FOLD Schritt 91 = (!E946 & E947 & !E948 + F285 & !E786 & E787 & !E788) & !F831 & A4039 + F836  ;%{SE}%MKUKATPVW %CVW_SPS %VST_CON %P 2:Schritt 91 = (!E946 & E947 & !E948 + F285 & !E786 & E787 & !E788) & !F831 & A4039 + F836 , 3: ST_CON
         IF (NOT $IN[946] AND $IN[947] AND NOT $IN[948] OR $FLAG[285] AND NOT $IN[786] AND $IN[787] AND NOT $IN[788]) AND NOT $FLAG[831] AND $OUT[4039] OR $FLAG[836] THEN
            PREVSTEP = $APP_INT[5]
            $APP_INT[5] = 91
         ENDIF
      ;ENDFOLD
   ;ENDFOLD
   ;FOLD SCHRITT 91 -- STAT EZ2/SP2/KE2 -- ;%{P}%MKUKATPVW,%CSTEP,%VST_NR,%P 1:SCHRITT, 2:91, 3: STAT EZ2/SP2/KE2
      ;FOLD ;%{H}
         Case 91
      ;ENDFOLD
      ;FOLD -- Hilfsflag SK Programmwechsel -- ;%{SE}%MKUKATPVW %CVW_COM %VCOMMENT %P 2:-- Hilfsflag SK Programmwechsel --, 3: VW_COMMENT
      ;ENDFOLD
      ;FOLD F334 = AUS ;%{SE}%MKUKATPVW %CVW_SPS %VBOASG %P 2:F334 = AUS, 3: BOASG
         $FLAG[334] = FALSE
      ;ENDFOLD
      ;FOLD -- RSK Sammelstoerung -- ;%{SE}%MKUKATPVW %CVW_COM %VCOMMENT %P 2:-- RSK Sammelstoerung --, 3: VW_COMMENT
      ;ENDFOLD
      ;FOLD F329 = T9 ;%{SE}%MKUKATPVW %CVW_SPS %VBOASG %P 2:F329 = T9, 3: BOASG
         $FLAG[329] = $TIMER_FLAG[9]
      ;ENDFOLD
      ;FOLD Schritt 92 = A4039 & E877 & (E917 & !E936 & !F831 + T9)  ;%{SE}%MKUKATPVW %CVW_SPS %VST_CON %P 2:Schritt 92 = A4039 & E877 & (E917 & !E936 & !F831 + T9) , 3: ST_CON
         IF $OUT[4039] AND $IN[877] AND ($IN[917] AND NOT $IN[936] AND NOT $FLAG[831] OR $TIMER_FLAG[9]) THEN
            PREVSTEP = $APP_INT[5]
            $APP_INT[5] = 92
         ENDIF
      ;ENDFOLD
      ;FOLD Schritt 92 = A4039 & E877 & (E885 & !E936 & F831 + T9)  ;%{SE}%MKUKATPVW %CVW_SPS %VST_CON %P 2:Schritt 92 = A4039 & E877 & (E885 & !E936 & F831 + T9) , 3: ST_CON
         IF $OUT[4039] AND $IN[877] AND ($IN[885] AND NOT $IN[936] AND $FLAG[831] OR $TIMER_FLAG[9]) THEN
            PREVSTEP = $APP_INT[5]
            $APP_INT[5] = 92
         ENDIF
      ;ENDFOLD
   ;ENDFOLD
   ;FOLD SCHRITT 92 -- STAT EZ2/SP2/KE2-- ;%{P}%MKUKATPVW,%CSTEP,%VST_NR,%P 1:SCHRITT, 2:92, 3: STAT EZ2/SP2/KE2
      ;FOLD ;%{H}
         Case 92
      ;ENDFOLD
      ;FOLD -- RSK Fehlerausgabe Kappenverschleiss -- ;%{SE}%MKUKATPVW %CVW_COM %VCOMMENT %P 2:-- RSK Fehlerausgabe Kappenverschleiss --, 3: VW_COMMENT
      ;ENDFOLD
      ;FOLD F160 = E937 ;%{SE}%MKUKATPVW %CVW_SPS %VBOASG %P 2:F160 = E937, 3: BOASG
         $FLAG[160] = $IN[937]
      ;ENDFOLD
      ;FOLD -- RSK Fehlerausgabe Messen -- ;%{SE}%MKUKATPVW %CVW_COM %VCOMMENT %P 2:-- RSK Fehlerausgabe Messen --, 3: VW_COMMENT
      ;ENDFOLD
      ;FOLD F326 = E936 + E937 + E938 + F326 ;%{SE}%MKUKATPVW %CVW_SPS %VBOASG %P 2:F326 = E936 + E937 + E938 + F326, 3: BOASG
         $FLAG[326] = $IN[936] OR $IN[937] OR $IN[938] OR $FLAG[326]
      ;ENDFOLD
      ;FOLD -- RSK Sammelstoerung -- ;%{SE}%MKUKATPVW %CVW_COM %VCOMMENT %P 2:-- RSK Sammelstoerung --, 3: VW_COMMENT
      ;ENDFOLD
      ;FOLD F329 = F326 ;%{SE}%MKUKATPVW %CVW_SPS %VBOASG %P 2:F329 = F326, 3: BOASG
         $FLAG[329] = $FLAG[326]
      ;ENDFOLD
      ;FOLD A918 = F831 & A918 ;%{SE}%MKUKATPVW %CVW_SPS %VBOASG %P 2:A918 = F831 & A918, 3: BOASG
         $OUT[918] = $FLAG[831] AND $OUT[918]
      ;ENDFOLD
      ;FOLD A919 = F831 & A919 ;%{SE}%MKUKATPVW %CVW_SPS %VBOASG %P 2:A919 = F831 & A919, 3: BOASG
         $OUT[919] = $FLAG[831] AND $OUT[919]
      ;ENDFOLD
      ;FOLD -- Hilfsflag Startfrasen EZ2/SP2 an SK1 -- ;%{SE}%MKUKATPVW %CVW_COM %VCOMMENT %P 2:-- Hilfsflag Startfrasen EZ2/SP2 an SK1 --, 3: VW_COMMENT
      ;ENDFOLD
      ;FOLD F307 = F285 & F138 & !F831 & !F830 ;%{SE}%MKUKATPVW %CVW_SPS %VBOASG %P 2:F307 = F285 & F138 & !F831 & !F830, 3: BOASG
         $FLAG[307] = $FLAG[285] AND $FLAG[138] AND NOT $FLAG[831] AND NOT $FLAG[830]
      ;ENDFOLD
      ;FOLD -- Hilfsflag Normalfrasen EZ2/SP2 an SK1 -- ;%{SE}%MKUKATPVW %CVW_COM %VCOMMENT %P 2:-- Hilfsflag Normalfrasen EZ2/SP2 an SK1 --, 3: VW_COMMENT
      ;ENDFOLD
      ;FOLD F308 = F285 & F139 & !F831 & !F830 ;%{SE}%MKUKATPVW %CVW_SPS %VBOASG %P 2:F308 = F285 & F139 & !F831 & !F830, 3: BOASG
         $FLAG[308] = $FLAG[285] AND $FLAG[139] AND NOT $FLAG[831] AND NOT $FLAG[830]
      ;ENDFOLD
      ;FOLD -- Ueberwachungszeit EZ2/SP2/KE2 Setzhub 2 -- ;%{SE}%MKUKATPVW %CVW_COM %VCOMMENT %P 2:-- Ueberwachungszeit EZ2/SP2/KE2 Setzhub 2 --, 3: VW_COMMENT
      ;ENDFOLD
      ;FOLD t9 ( EIN ) = -80[1/10Sek] ;%{SE}%MKUKATPVW %CVW_SPS %VTASG %P 2:t9 ( EIN ) = -80[1/10Sek], 3: TASG
         VW(#SET_TIME,TRUE,9,0,-80)
      ;ENDFOLD
      ;FOLD -- Druckvorgabe SK2/SK1/EZ2/SP2/KE2 -- ;%{SE}%MKUKATPVW %CVW_COM %VCOMMENT %P 2:-- Druckvorgabe SK2/SK1/EZ2/SP2/KE2 --, 3: VW_COMMENT
      ;ENDFOLD
      ;FOLD bin3 (F307) = 45 ;%{SE}%MKUKATPVW %CVW_SPS %VARIASG %P 2:bin3 (F307) = 45, 3: ARIASG
         VW(#BINOUT,$FLAG[307],3,45)
      ;ENDFOLD
      ;FOLD bin3 (F308) = 55 ;%{SE}%MKUKATPVW %CVW_SPS %VARIASG %P 2:bin3 (F308) = 55, 3: ARIASG
         VW(#BINOUT,$FLAG[308],3,55)
      ;ENDFOLD
      ;FOLD bin4 (F138) = 41 ;%{SE}%MKUKATPVW %CVW_SPS %VARIASG %P 2:bin4 (F138) = 41, 3: ARIASG
         VW(#BINOUT,$FLAG[138],4,41)
      ;ENDFOLD
      ;FOLD bin4 (F139) = 51 ;%{SE}%MKUKATPVW %CVW_SPS %VARIASG %P 2:bin4 (F139) = 51, 3: ARIASG
         VW(#BINOUT,$FLAG[139],4,51)
      ;ENDFOLD
      ;FOLD bin6 (F138) = 41 ;%{SE}%MKUKATPVW %CVW_SPS %VARIASG %P 2:bin6 (F138) = 41, 3: ARIASG
         VW(#BINOUT,$FLAG[138],6,41)
      ;ENDFOLD
      ;FOLD bin6 (F139) = 51 ;%{SE}%MKUKATPVW %CVW_SPS %VARIASG %P 2:bin6 (F139) = 51, 3: ARIASG
         VW(#BINOUT,$FLAG[139],6,51)
      ;ENDFOLD
      ;FOLD -- Wartezeit Programmwechsel SK -- ;%{SE}%MKUKATPVW %CVW_COM %VCOMMENT %P 2:-- Wartezeit Programmwechsel SK --, 3: VW_COMMENT
      ;ENDFOLD
      ;FOLD T8 ( !F334 ) = -2[1/10Sek] ;%{SE}%MKUKATPVW %CVW_SPS %VTASG %P 2:T8 ( !F334 ) = -2[1/10Sek], 3: TASG
         VW(#SET_TIME,NOT $FLAG[334],8,0,-2)
      ;ENDFOLD
      ;FOLD -- Hilfsflag SK Programmwechsel -- ;%{SE}%MKUKATPVW %CVW_COM %VCOMMENT %P 2:-- Hilfsflag SK Programmwechsel --, 3: VW_COMMENT
      ;ENDFOLD
      ;FOLD F334 = EIN ;%{SE}%MKUKATPVW %CVW_SPS %VBOASG %P 2:F334 = EIN, 3: BOASG
         $FLAG[334] = TRUE
      ;ENDFOLD
      ;FOLD Schritt 93 = T8 & !F335 & A4039  ;%{SE}%MKUKATPVW %CVW_SPS %VST_CON %P 2:Schritt 93 = T8 & !F335 & A4039 , 3: ST_CON
         IF $TIMER_FLAG[8] AND NOT $FLAG[335] AND $OUT[4039] THEN
            PREVSTEP = $APP_INT[5]
            $APP_INT[5] = 93
         ENDIF
      ;ENDFOLD
      ;FOLD Schritt 93 = T8 & F335 & !F138 & !F307 & A4039  ;%{SE}%MKUKATPVW %CVW_SPS %VST_CON %P 2:Schritt 93 = T8 & F335 & !F138 & !F307 & A4039 , 3: ST_CON
         IF $TIMER_FLAG[8] AND $FLAG[335] AND NOT $FLAG[138] AND NOT $FLAG[307] AND $OUT[4039] THEN
            PREVSTEP = $APP_INT[5]
            $APP_INT[5] = 93
         ENDIF
      ;ENDFOLD
      ;FOLD Schritt 222 = T8 & F335 & (F307 + F138) & A4039  ;%{SE}%MKUKATPVW %CVW_SPS %VST_CON %P 2:Schritt 222 = T8 & F335 & (F307 + F138) & A4039 , 3: ST_CON
         IF $TIMER_FLAG[8] AND $FLAG[335] AND ($FLAG[307] OR $FLAG[138]) AND $OUT[4039] THEN
            PREVSTEP = $APP_INT[5]
            $APP_INT[5] = 222
         ENDIF
      ;ENDFOLD
   ;ENDFOLD
   ;FOLD SCHRITT 93 -- STAT EZ2/SP2/KE2 -- ;%{P}%MKUKATPVW,%CSTEP,%VST_NR,%P 1:SCHRITT, 2:93, 3: STAT EZ2/SP2/KE2
      ;FOLD ;%{H}
         Case 93
      ;ENDFOLD
      ;FOLD -- Hilfsflag SK Programmwechsel -- ;%{SE}%MKUKATPVW %CVW_COM %VCOMMENT %P 2:-- Hilfsflag SK Programmwechsel --, 3: VW_COMMENT
      ;ENDFOLD
      ;FOLD F334 = AUS ;%{SE}%MKUKATPVW %CVW_SPS %VBOASG %P 2:F334 = AUS, 3: BOASG
         $FLAG[334] = FALSE
      ;ENDFOLD
      ;FOLD A917 = F831 & A917 ;%{SE}%MKUKATPVW %CVW_SPS %VBOASG %P 2:A917 = F831 & A917, 3: BOASG
         $OUT[917] = $FLAG[831] AND $OUT[917]
      ;ENDFOLD
      ;FOLD -- EZ2/SP2/KE2 schliessen -- ;%{SE}%MKUKATPVW %CVW_COM %VCOMMENT %P 2:-- EZ2/SP2/KE2 schliessen --, 3: VW_COMMENT
      ;ENDFOLD
      ;FOLD A885 = !F831 & A885 ;%{SE}%MKUKATPVW %CVW_SPS %VBOASG %P 2:A885 = !F831 & A885, 3: BOASG
         $OUT[885] = NOT $FLAG[831] AND $OUT[885]
      ;ENDFOLD
      ;FOLD A877 = AUS ;%{SE}%MKUKATPVW %CVW_SPS %VBOASG %P 2:A877 = AUS, 3: BOASG
         $OUT[877] = FALSE
      ;ENDFOLD
      ;FOLD A878 = !F329 & !F160 ;%{SE}%MKUKATPVW %CVW_SPS %VBOASG %P 2:A878 = !F329 & !F160, 3: BOASG
         $OUT[878] = NOT $FLAG[329] AND NOT $FLAG[160]
      ;ENDFOLD
      ;FOLD -- Ueberwachungszeit Kurzschlussschweissung SK2/SK1 -- ;%{SE}%MKUKATPVW %CVW_COM %VCOMMENT %P 2:-- Ueberwachungszeit Kurzschlussschweissung SK2/SK1 --, 3: VW_COMMENT
      ;ENDFOLD
      ;FOLD t9 ( EIN ) = -80[1/10Sek] ;%{SE}%MKUKATPVW %CVW_SPS %VTASG %P 2:t9 ( EIN ) = -80[1/10Sek], 3: TASG
         VW(#SET_TIME,TRUE,9,0,-80)
      ;ENDFOLD
      ;FOLD Schritt 94 = F285 & A514 & !E877 & E878 + E877 & !E878 & (F329 + F326 + F160) & A4039  ;%{SE}%MKUKATPVW %CVW_SPS %VST_CON %P 2:Schritt 94 = F285 & A514 & !E877 & E878 + E877 & !E878 & (F329 + F326 + F160) & A4039 , 3: ST_CON
         IF $FLAG[285] AND $OUT[514] AND NOT $IN[877] AND $IN[878] OR $IN[877] AND NOT $IN[878] AND ($FLAG[329] OR $FLAG[326] OR $FLAG[160]) AND $OUT[4039] THEN
            PREVSTEP = $APP_INT[5]
            $APP_INT[5] = 94
         ENDIF
      ;ENDFOLD
      ;FOLD Schritt 94 = !F285 & !A514 & !E877 & E878 + E877 & !E878 & (F329 + F326 + F160) & A4039  ;%{SE}%MKUKATPVW %CVW_SPS %VST_CON %P 2:Schritt 94 = !F285 & !A514 & !E877 & E878 + E877 & !E878 & (F329 + F326 + F160) & A4039 , 3: ST_CON
         IF NOT $FLAG[285] AND NOT $OUT[514] AND NOT $IN[877] AND $IN[878] OR $IN[877] AND NOT $IN[878] AND ($FLAG[329] OR $FLAG[326] OR $FLAG[160]) AND $OUT[4039] THEN
            PREVSTEP = $APP_INT[5]
            $APP_INT[5] = 94
         ENDIF
      ;ENDFOLD
   ;ENDFOLD
   ;FOLD SCHRITT 94 -- STAT EZ2/SP2/KE2-- ;%{P}%MKUKATPVW,%CSTEP,%VST_NR,%P 1:SCHRITT, 2:94, 3: STAT EZ2/SP2/KE2
      ;FOLD ;%{H}
         Case 94
      ;ENDFOLD
      ;FOLD -- Hilfsflag SK Programmwechsel -- ;%{SE}%MKUKATPVW %CVW_COM %VCOMMENT %P 2:-- Hilfsflag SK Programmwechsel --, 3: VW_COMMENT
      ;ENDFOLD
      ;FOLD F334 = AUS ;%{SE}%MKUKATPVW %CVW_SPS %VBOASG %P 2:F334 = AUS, 3: BOASG
         $FLAG[334] = FALSE
      ;ENDFOLD
      ;FOLD t9 ( EIN ) = STOP ;%{SE}%MKUKATPVW %CVW_SPS %VTSTOP %P 2:t9 ( EIN ) = STOP, 3: TSTOP
         VW(#SET_TIME,TRUE,9,1,0)
      ;ENDFOLD
      ;FOLD -- RSK Fehlerausgabe EZ2/SP2/KE2 Kraftaufbau -- ;%{SE}%MKUKATPVW %CVW_COM %VCOMMENT %P 2:-- RSK Fehlerausgabe EZ2/SP2/KE2 Kraftaufbau --, 3: VW_COMMENT
      ;ENDFOLD
      ;FOLD F325 = T9 + F325 ;%{SE}%MKUKATPVW %CVW_SPS %VBOASG %P 2:F325 = T9 + F325, 3: BOASG
         $FLAG[325] = $TIMER_FLAG[9] OR $FLAG[325]
      ;ENDFOLD
      ;FOLD -- RSK Fehlerausgabe K -- ;%{SE}%MKUKATPVW %CVW_COM %VCOMMENT %P 2:-- RSK Fehlerausgabe K --, 3: VW_COMMENT
      ;ENDFOLD
      ;FOLD F836 = (A945 & E965 + A945 & !E962) + (A785 & E805 + A785 & !E802) ;%{SE}%MKUKATPVW %CVW_SPS %VBOASG %P 2:F836 = (A945 & E965 + A945 & !E962) + (A785 & E805 + A785 & !E802), 3: BOASG
         $FLAG[836] = ($OUT[945] AND $IN[965] OR $OUT[945] AND NOT $IN[962]) OR ($OUT[785] AND $IN[805] OR $OUT[785] AND NOT $IN[802])
      ;ENDFOLD
      ;FOLD F327 = (F836 & !F831) + (F831 & A878 & E948 + A878 & !E865) + F327 ;%{SE}%MKUKATPVW %CVW_SPS %VBOASG %P 2:F327 = (F836 & !F831) + (F831 & A878 & E948 + A878 & !E865) + F327, 3: BOASG
         $FLAG[327] = ($FLAG[836] AND NOT $FLAG[831]) OR ($FLAG[831] AND $OUT[878] AND $IN[948] OR $OUT[878] AND NOT $IN[865]) OR $FLAG[327]
      ;ENDFOLD
      ;FOLD -- RSK Sammelstoerung -- ;%{SE}%MKUKATPVW %CVW_COM %VCOMMENT %P 2:-- RSK Sammelstoerung --, 3: VW_COMMENT
      ;ENDFOLD
      ;FOLD F329 = F325 + F326 + F327 ;%{SE}%MKUKATPVW %CVW_SPS %VBOASG %P 2:F329 = F325 + F326 + F327, 3: BOASG
         $FLAG[329] = $FLAG[325] OR $FLAG[326] OR $FLAG[327]
      ;ENDFOLD
      ;FOLD A192 = !F285 & F329 ;%{SE}%MKUKATPVW %CVW_SPS %VBOASG %P 2:A192 = !F285 & F329, 3: BOASG
         $OUT[192] = NOT $FLAG[285] AND $FLAG[329]
      ;ENDFOLD
      ;FOLD A160 = F285 & F329 & !F831 & !F830 ;%{SE}%MKUKATPVW %CVW_SPS %VBOASG %P 2:A160 = F285 & F329 & !F831 & !F830, 3: BOASG
         $OUT[160] = $FLAG[285] AND $FLAG[329] AND NOT $FLAG[831] AND NOT $FLAG[830]
      ;ENDFOLD
      ;FOLD -- Kurzschlussschweissung SK2/SK1 -- ;%{SE}%MKUKATPVW %CVW_COM %VCOMMENT %P 2:-- Kurzschlussschweissung SK2/SK1 --, 3: VW_COMMENT
      ;ENDFOLD
      ;FOLD F836 = AUS ;%{SE}%MKUKATPVW %CVW_SPS %VBOASG %P 2:F836 = AUS, 3: BOASG
         $FLAG[836] = FALSE
      ;ENDFOLD
      ;FOLD A945 = (!F285 & !F325 & !F329 & !F160 & !F831) + (F831 & A945) ;%{SE}%MKUKATPVW %CVW_SPS %VBOASG %P 2:A945 = (!F285 & !F325 & !F329 & !F160 & !F831) + (F831 & A945), 3: BOASG
         $OUT[945] = (NOT $FLAG[285] AND NOT $FLAG[325] AND NOT $FLAG[329] AND NOT $FLAG[160] AND NOT $FLAG[831]) OR ($FLAG[831] AND $OUT[945])
      ;ENDFOLD
      ;FOLD A785 = (F285 & !F325 & !F329 & !F160 + !F285 & A785) & !F831 & !F830 ;%{SE}%MKUKATPVW %CVW_SPS %VBOASG %P 2:A785 = (F285 & !F325 & !F329 & !F160 + !F285 & A785) & !F831 & !F830, 3: BOASG
         $OUT[785] = ($FLAG[285] AND NOT $FLAG[325] AND NOT $FLAG[329] AND NOT $FLAG[160] OR NOT $FLAG[285] AND $OUT[785]) AND NOT $FLAG[831] AND NOT $FLAG[830]
      ;ENDFOLD
      ;FOLD A878 = (!F285 & !F325 & !F329 & !F160 & F831) + (!F831 & A878) ;%{SE}%MKUKATPVW %CVW_SPS %VBOASG %P 2:A878 = (!F285 & !F325 & !F329 & !F160 & F831) + (!F831 & A878), 3: BOASG
         $OUT[878] = (NOT $FLAG[285] AND NOT $FLAG[325] AND NOT $FLAG[329] AND NOT $FLAG[160] AND $FLAG[831]) OR (NOT $FLAG[831] AND $OUT[878])
      ;ENDFOLD
      ;FOLD F836 = F326 + F327 + F160 ;%{SE}%MKUKATPVW %CVW_SPS %VBOASG %P 2:F836 = F326 + F327 + F160, 3: BOASG
         $FLAG[836] = $FLAG[326] OR $FLAG[327] OR $FLAG[160]
      ;ENDFOLD
      ;FOLD -- Flagbildung Wiederholfraesen -- ;%{SE}%MKUKATPVW %CVW_COM %VCOMMENT %P 2:-- Flagbildung Wiederholfraesen --, 3: VW_COMMENT
      ;ENDFOLD
      ;FOLD F749 = (F322 + F323 + F325 + F326 + F327 + F329) & !F748 ;%{SE}%MKUKATPVW %CVW_SPS %VBOASG %P 2:F749 = (F322 + F323 + F325 + F326 + F327 + F329) & !F748, 3: BOASG
         $FLAG[749] = ($FLAG[322] OR $FLAG[323] OR $FLAG[325] OR $FLAG[326] OR $FLAG[327] OR $FLAG[329]) AND NOT $FLAG[748]
      ;ENDFOLD
      ;FOLD Schritt 95 = (!F285 & E945 & E964 & !F831 + F285 & E785 & E804 & !F831 + F836) & A4039  ;%{SE}%MKUKATPVW %CVW_SPS %VST_CON %P 2:Schritt 95 = (!F285 & E945 & E964 & !F831 + F285 & E785 & E804 & !F831 + F836) & A4039 , 3: ST_CON
         IF (NOT $FLAG[285] AND $IN[945] AND $IN[964] AND NOT $FLAG[831] OR $FLAG[285] AND $IN[785] AND $IN[804] AND NOT $FLAG[831] OR $FLAG[836]) AND $OUT[4039] THEN
            PREVSTEP = $APP_INT[5]
            $APP_INT[5] = 95
         ENDIF
      ;ENDFOLD
      ;FOLD Schritt 95 = (!F285 & E945 & E15 & !F831 + F285 & E785 & E15 & !F831 + F836) & A4039  ;%{SE}%MKUKATPVW %CVW_SPS %VST_CON %P 2:Schritt 95 = (!F285 & E945 & E15 & !F831 + F285 & E785 & E15 & !F831 + F836) & A4039 , 3: ST_CON
         IF (NOT $FLAG[285] AND $IN[945] AND $IN[15] AND NOT $FLAG[831] OR $FLAG[285] AND $IN[785] AND $IN[15] AND NOT $FLAG[831] OR $FLAG[836]) AND $OUT[4039] THEN
            PREVSTEP = $APP_INT[5]
            $APP_INT[5] = 95
         ENDIF
      ;ENDFOLD
      ;FOLD Schritt 95 = (!F285 & E879 & E947 & F831 + F836) & A4039  ;%{SE}%MKUKATPVW %CVW_SPS %VST_CON %P 2:Schritt 95 = (!F285 & E879 & E947 & F831 + F836) & A4039 , 3: ST_CON
         IF (NOT $FLAG[285] AND $IN[879] AND $IN[947] AND $FLAG[831] OR $FLAG[836]) AND $OUT[4039] THEN
            PREVSTEP = $APP_INT[5]
            $APP_INT[5] = 95
         ENDIF
      ;ENDFOLD
      ;FOLD Schritt 95 = (!F285 & E879 & E15 & F831 + F836) & A4039  ;%{SE}%MKUKATPVW %CVW_SPS %VST_CON %P 2:Schritt 95 = (!F285 & E879 & E15 & F831 + F836) & A4039 , 3: ST_CON
         IF (NOT $FLAG[285] AND $IN[879] AND $IN[15] AND $FLAG[831] OR $FLAG[836]) AND $OUT[4039] THEN
            PREVSTEP = $APP_INT[5]
            $APP_INT[5] = 95
         ENDIF
      ;ENDFOLD
   ;ENDFOLD
   ;FOLD SCHRITT 95 -- STAT EZ2/SP2/KE2 -- ;%{P}%MKUKATPVW,%CSTEP,%VST_NR,%P 1:SCHRITT, 2:95, 3: STAT EZ2/SP2/KE2
      ;FOLD ;%{H}
         Case 95
      ;ENDFOLD
      ;FOLD F836 = AUS ;%{SE}%MKUKATPVW %CVW_SPS %VBOASG %P 2:F836 = AUS, 3: BOASG
         $FLAG[836] = FALSE
      ;ENDFOLD
      ;FOLD A945 = F831 & A945 ;%{SE}%MKUKATPVW %CVW_SPS %VBOASG %P 2:A945 = F831 & A945, 3: BOASG
         $OUT[945] = $FLAG[831] AND $OUT[945]
      ;ENDFOLD
      ;FOLD A785 = F285 & !E785 & !F831 & !F830 + !F285 & A785 & !F831 & !F830 ;%{SE}%MKUKATPVW %CVW_SPS %VBOASG %P 2:A785 = F285 & !E785 & !F831 & !F830 + !F285 & A785 & !F831 & !F830, 3: BOASG
         $OUT[785] = $FLAG[285] AND NOT $IN[785] AND NOT $FLAG[831] AND NOT $FLAG[830] OR NOT $FLAG[285] AND $OUT[785] AND NOT $FLAG[831] AND NOT $FLAG[830]
      ;ENDFOLD
      ;FOLD F138 = !F327 & F138 ;%{SE}%MKUKATPVW %CVW_SPS %VBOASG %P 2:F138 = !F327 & F138, 3: BOASG
         $FLAG[138] = NOT $FLAG[327] AND $FLAG[138]
      ;ENDFOLD
      ;FOLD F139 = F327 + F139 ;%{SE}%MKUKATPVW %CVW_SPS %VBOASG %P 2:F139 = F327 + F139, 3: BOASG
         $FLAG[139] = $FLAG[327] OR $FLAG[139]
      ;ENDFOLD
      ;FOLD -- EZ2/SP2/KE2 oeffnen -- ;%{SE}%MKUKATPVW %CVW_COM %VCOMMENT %P 2:-- EZ2/SP2/KE2 oeffnen --, 3: VW_COMMENT
      ;ENDFOLD
      ;FOLD A879 = AUS ;%{SE}%MKUKATPVW %CVW_SPS %VBOASG %P 2:A879 = AUS, 3: BOASG
         $OUT[879] = FALSE
      ;ENDFOLD
      ;FOLD A878 = AUS ;%{SE}%MKUKATPVW %CVW_SPS %VBOASG %P 2:A878 = AUS, 3: BOASG
         $OUT[878] = FALSE
      ;ENDFOLD
      ;FOLD A877 = !E877 ;%{SE}%MKUKATPVW %CVW_SPS %VBOASG %P 2:A877 = !E877, 3: BOASG
         $OUT[877] = NOT $IN[877]
      ;ENDFOLD
      ;FOLD -- Hilfflag fuer KE 2 -- ;%{SE}%MKUKATPVW %CVW_COM %VCOMMENT %P 2:-- Hilfflag fuer KE 2 --, 3: VW_COMMENT
      ;ENDFOLD
      ;FOLD F836 = !F285 & !F831 ;%{SE}%MKUKATPVW %CVW_SPS %VBOASG %P 2:F836 = !F285 & !F831, 3: BOASG
         $FLAG[836] = NOT $FLAG[285] AND NOT $FLAG[831]
      ;ENDFOLD
      ;FOLD bin3 (F285) = 5 ;%{SE}%MKUKATPVW %CVW_SPS %VARIASG %P 2:bin3 (F285) = 5, 3: ARIASG
         VW(#BINOUT,$FLAG[285],3,5)
      ;ENDFOLD
      ;FOLD bin6 (F836) = 1 ;%{SE}%MKUKATPVW %CVW_SPS %VARIASG %P 2:bin6 (F836) = 1, 3: ARIASG
         VW(#BINOUT,$FLAG[836],6,1)
      ;ENDFOLD
      ;FOLD -- Wartezeit Programmwechsel SK -- ;%{SE}%MKUKATPVW %CVW_COM %VCOMMENT %P 2:-- Wartezeit Programmwechsel SK --, 3: VW_COMMENT
      ;ENDFOLD
      ;FOLD T8 ( !F334 ) = -2[1/10Sek] ;%{SE}%MKUKATPVW %CVW_SPS %VTASG %P 2:T8 ( !F334 ) = -2[1/10Sek], 3: TASG
         VW(#SET_TIME,NOT $FLAG[334],8,0,-2)
      ;ENDFOLD
      ;FOLD -- Hilfsflag SK Programmwechsel -- ;%{SE}%MKUKATPVW %CVW_COM %VCOMMENT %P 2:-- Hilfsflag SK Programmwechsel --, 3: VW_COMMENT
      ;ENDFOLD
      ;FOLD F334 = EIN ;%{SE}%MKUKATPVW %CVW_SPS %VBOASG %P 2:F334 = EIN, 3: BOASG
         $FLAG[334] = TRUE
      ;ENDFOLD
      ;FOLD F748 = F322 + F323 + F325 + F326 + F327 + F329 ;%{SE}%MKUKATPVW %CVW_SPS %VBOASG %P 2:F748 = F322 + F323 + F325 + F326 + F327 + F329, 3: BOASG
         $FLAG[748] = $FLAG[322] OR $FLAG[323] OR $FLAG[325] OR $FLAG[326] OR $FLAG[327] OR $FLAG[329]
      ;ENDFOLD
      ;FOLD Schritt 74 = E877 & !E878 & (F322 + F323 + F325 + F326 + F327 + F329) & (E26 + E27) & A4039  ;%{SE}%MKUKATPVW %CVW_SPS %VST_CON %P 2:Schritt 74 = E877 & !E878 & (F322 + F323 + F325 + F326 + F327 + F329) & (E26 + E27) & A4039 , 3: ST_CON
         IF $IN[877] AND NOT $IN[878] AND ($FLAG[322] OR $FLAG[323] OR $FLAG[325] OR $FLAG[326] OR $FLAG[327] OR $FLAG[329]) AND ($IN[26] OR $IN[27]) AND $OUT[4039] THEN
            PREVSTEP = $APP_INT[5]
            $APP_INT[5] = 74
         ENDIF
      ;ENDFOLD
      ;FOLD Schritt 74 = E877 & !E878 & (F322 + F323 + F325 + F326 + F327 + F329) & (F731 & F749) & A4039  ;%{SE}%MKUKATPVW %CVW_SPS %VST_CON %P 2:Schritt 74 = E877 & !E878 & (F322 + F323 + F325 + F326 + F327 + F329) & (F731 & F749) & A4039 , 3: ST_CON
         IF $IN[877] AND NOT $IN[878] AND ($FLAG[322] OR $FLAG[323] OR $FLAG[325] OR $FLAG[326] OR $FLAG[327] OR $FLAG[329]) AND ($FLAG[731] AND $FLAG[749]) AND $OUT[4039] THEN
            PREVSTEP = $APP_INT[5]
            $APP_INT[5] = 74
         ENDIF
      ;ENDFOLD
      ;FOLD Schritt 96 = T8 & E877 & !E878 & (!F325 & !F326 & !F327 & !F329 + F160) & A4039  ;%{SE}%MKUKATPVW %CVW_SPS %VST_CON %P 2:Schritt 96 = T8 & E877 & !E878 & (!F325 & !F326 & !F327 & !F329 + F160) & A4039 , 3: ST_CON
         IF $TIMER_FLAG[8] AND $IN[877] AND NOT $IN[878] AND (NOT $FLAG[325] AND NOT $FLAG[326] AND NOT $FLAG[327] AND NOT $FLAG[329] OR $FLAG[160]) AND $OUT[4039] THEN
            PREVSTEP = $APP_INT[5]
            $APP_INT[5] = 96
         ENDIF
      ;ENDFOLD
   ;ENDFOLD
   ;FOLD SCHRITT 96 -- STAT EZ2/SP2/KE2 # Ende -- ;%{P}%MKUKATPVW,%CSTEP,%VST_NR,%P 1:SCHRITT, 2:96, 3: STAT EZ2/SP2/KE2 # Ende
      ;FOLD ;%{H}
         Case 96
      ;ENDFOLD
      ;FOLD -- Hilfsflag SK Programmwechsel -- ;%{SE}%MKUKATPVW %CVW_COM %VCOMMENT %P 2:-- Hilfsflag SK Programmwechsel --, 3: VW_COMMENT
      ;ENDFOLD
      ;FOLD F334 = AUS ;%{SE}%MKUKATPVW %CVW_SPS %VBOASG %P 2:F334 = AUS, 3: BOASG
         $FLAG[334] = FALSE
      ;ENDFOLD
      ;FOLD A116 = AUS ;%{SE}%MKUKATPVW %CVW_SPS %VBOASG %P 2:A116 = AUS, 3: BOASG
         $OUT[116] = FALSE
      ;ENDFOLD
      ;FOLD A162 = AUS ;%{SE}%MKUKATPVW %CVW_SPS %VBOASG %P 2:A162 = AUS, 3: BOASG
         $OUT[162] = FALSE
      ;ENDFOLD
      ;FOLD F836 = AUS ;%{SE}%MKUKATPVW %CVW_SPS %VBOASG %P 2:F836 = AUS, 3: BOASG
         $FLAG[836] = FALSE
      ;ENDFOLD
      ;FOLD F836 = (!F285 & !E946 & E947 &!E948 + F285 & !E786 & E787 & !E788) & !F831 ;%{SE}%MKUKATPVW %CVW_SPS %VBOASG %P 2:F836 = (!F285 & !E946 & E947 &!E948 + F285 & !E786 & E787 & !E788) & !F831, 3: BOASG
         $FLAG[836] = (NOT $FLAG[285] AND NOT $IN[946] AND $IN[947] AND NOT $IN[948] OR $FLAG[285] AND NOT $IN[786] AND $IN[787] AND NOT $IN[788]) AND NOT $FLAG[831]
      ;ENDFOLD
      ;FOLD -- RSK Sammelstoerung -- ;%{SE}%MKUKATPVW %CVW_COM %VCOMMENT %P 2:-- RSK Sammelstoerung --, 3: VW_COMMENT
      ;ENDFOLD
      ;FOLD F329 = F160 ;%{SE}%MKUKATPVW %CVW_SPS %VBOASG %P 2:F329 = F160, 3: BOASG
         $FLAG[329] = $FLAG[160]
      ;ENDFOLD
      ;FOLD F149 = (!E881 & !E883 & F831) + F836 & !F831 + F160 & (E26 + E27) ;%{SE}%MKUKATPVW %CVW_SPS %VBOASG %P 2:F149 = (!E881 & !E883 & F831) + F836 & !F831 + F160 & (E26 + E27), 3: BOASG
         $FLAG[149] = (NOT $IN[881] AND NOT $IN[883] AND $FLAG[831]) OR $FLAG[836] AND NOT $FLAG[831] OR $FLAG[160] AND ($IN[26] OR $IN[27])
      ;ENDFOLD
      ;FOLD Schritt 1 = F149 & A4039  ;%{SE}%MKUKATPVW %CVW_SPS %VST_CON %P 2:Schritt 1 = F149 & A4039 , 3: ST_CON
         IF $FLAG[149] AND $OUT[4039] THEN
            PREVSTEP = $APP_INT[5]
            $APP_INT[5] = 1
         ENDIF
      ;ENDFOLD
   ;ENDFOLD
   ;FOLD SCHRITT 97 -- STAT EZ3/SP3/KE3 # Start -- ;%{P}%MKUKATPVW,%CSTEP,%VST_NR,%P 1:SCHRITT, 2:97, 3: STAT EZ3/SP3/KE3 # Start
      ;FOLD ;%{H}
         Case 97
      ;ENDFOLD
      ;FOLD -- RSK gestartet -- ;%{SE}%MKUKATPVW %CVW_COM %VCOMMENT %P 2:-- RSK gestartet --, 3: VW_COMMENT
      ;ENDFOLD
      ;FOLD F196 = AUS ;%{SE}%MKUKATPVW %CVW_SPS %VBOASG %P 2:F196 = AUS, 3: BOASG
         $FLAG[196] = FALSE
      ;ENDFOLD
      ;FOLD F321 = AUS ;%{SE}%MKUKATPVW %CVW_SPS %VBOASG %P 2:F321 = AUS, 3: BOASG
         $FLAG[321] = FALSE
      ;ENDFOLD
      ;FOLD F322 = AUS ;%{SE}%MKUKATPVW %CVW_SPS %VBOASG %P 2:F322 = AUS, 3: BOASG
         $FLAG[322] = FALSE
      ;ENDFOLD
      ;FOLD F323 = AUS ;%{SE}%MKUKATPVW %CVW_SPS %VBOASG %P 2:F323 = AUS, 3: BOASG
         $FLAG[323] = FALSE
      ;ENDFOLD
      ;FOLD F324 = AUS ;%{SE}%MKUKATPVW %CVW_SPS %VBOASG %P 2:F324 = AUS, 3: BOASG
         $FLAG[324] = FALSE
      ;ENDFOLD
      ;FOLD F325 = AUS ;%{SE}%MKUKATPVW %CVW_SPS %VBOASG %P 2:F325 = AUS, 3: BOASG
         $FLAG[325] = FALSE
      ;ENDFOLD
      ;FOLD F326 = AUS ;%{SE}%MKUKATPVW %CVW_SPS %VBOASG %P 2:F326 = AUS, 3: BOASG
         $FLAG[326] = FALSE
      ;ENDFOLD
      ;FOLD F327 = AUS ;%{SE}%MKUKATPVW %CVW_SPS %VBOASG %P 2:F327 = AUS, 3: BOASG
         $FLAG[327] = FALSE
      ;ENDFOLD
      ;FOLD F329 = AUS ;%{SE}%MKUKATPVW %CVW_SPS %VBOASG %P 2:F329 = AUS, 3: BOASG
         $FLAG[329] = FALSE
      ;ENDFOLD
      ;FOLD -- EZ3/SP3/KE3 Zaehler -- ;%{SE}%MKUKATPVW %CVW_COM %VCOMMENT %P 2:-- EZ3/SP3/KE3 Zaehler --, 3: VW_COMMENT
      ;ENDFOLD
      ;FOLD F186 = AUS ;%{SE}%MKUKATPVW %CVW_SPS %VBOASG %P 2:F186 = AUS, 3: BOASG
         $FLAG[186] = FALSE
      ;ENDFOLD
      ;FOLD F187 = AUS ;%{SE}%MKUKATPVW %CVW_SPS %VBOASG %P 2:F187 = AUS, 3: BOASG
         $FLAG[187] = FALSE
      ;ENDFOLD
      ;FOLD F188 = AUS ;%{SE}%MKUKATPVW %CVW_SPS %VBOASG %P 2:F188 = AUS, 3: BOASG
         $FLAG[188] = FALSE
      ;ENDFOLD
      ;FOLD F189 = AUS ;%{SE}%MKUKATPVW %CVW_SPS %VBOASG %P 2:F189 = AUS, 3: BOASG
         $FLAG[189] = FALSE
      ;ENDFOLD
      ;FOLD F190 = AUS ;%{SE}%MKUKATPVW %CVW_SPS %VBOASG %P 2:F190 = AUS, 3: BOASG
         $FLAG[190] = FALSE
      ;ENDFOLD
      ;FOLD F191 = AUS ;%{SE}%MKUKATPVW %CVW_SPS %VBOASG %P 2:F191 = AUS, 3: BOASG
         $FLAG[191] = FALSE
      ;ENDFOLD
      ;FOLD -- Hilfsflags Funktionstest KF Motor -- ;%{SE}%MKUKATPVW %CVW_COM %VCOMMENT %P 2:-- Hilfsflags Funktionstest KF Motor --, 3: VW_COMMENT
      ;ENDFOLD
      ;FOLD F312 = AUS ;%{SE}%MKUKATPVW %CVW_SPS %VBOASG %P 2:F312 = AUS, 3: BOASG
         $FLAG[312] = FALSE
      ;ENDFOLD
      ;FOLD F313 = AUS ;%{SE}%MKUKATPVW %CVW_SPS %VBOASG %P 2:F313 = AUS, 3: BOASG
         $FLAG[313] = FALSE
      ;ENDFOLD
      ;FOLD bin7 ( EIN ) = 31 ;%{SE}%MKUKATPVW %CVW_SPS %VARIASG %P 2:bin7 ( EIN ) = 31, 3: ARIASG
         VW(#BINOUT,TRUE,7,31)
      ;ENDFOLD
      ;FOLD bin9 ( EIN ) = 31 ;%{SE}%MKUKATPVW %CVW_SPS %VARIASG %P 2:bin9 ( EIN ) = 31, 3: ARIASG
         VW(#BINOUT,TRUE,9,31)
      ;ENDFOLD
      ;FOLD -- Wartezeit Programmwechsel SK -- ;%{SE}%MKUKATPVW %CVW_COM %VCOMMENT %P 2:-- Wartezeit Programmwechsel SK --, 3: VW_COMMENT
      ;ENDFOLD
      ;FOLD T8 ( !F334 ) = -2[1/10Sek] ;%{SE}%MKUKATPVW %CVW_SPS %VTASG %P 2:T8 ( !F334 ) = -2[1/10Sek], 3: TASG
         VW(#SET_TIME,NOT $FLAG[334],8,0,-2)
      ;ENDFOLD
      ;FOLD -- Hilfsflag SK Programmwechsel -- ;%{SE}%MKUKATPVW %CVW_COM %VCOMMENT %P 2:-- Hilfsflag SK Programmwechsel --, 3: VW_COMMENT
      ;ENDFOLD
      ;FOLD F334 = EIN ;%{SE}%MKUKATPVW %CVW_SPS %VBOASG %P 2:F334 = EIN, 3: BOASG
         $FLAG[334] = TRUE
      ;ENDFOLD
      ;FOLD -- Stat. EZ3/SP3/KE3 beim Fraesen -- ;%{SE}%MKUKATPVW %CVW_COM %VCOMMENT %P 2:-- Stat. EZ3/SP3/KE3 beim Fraesen --, 3: VW_COMMENT
      ;ENDFOLD
      ;FOLD A116 = EIN ;%{SE}%MKUKATPVW %CVW_SPS %VBOASG %P 2:A116 = EIN, 3: BOASG
         $OUT[116] = TRUE
      ;ENDFOLD
      ;FOLD A194 = EIN ;%{SE}%MKUKATPVW %CVW_SPS %VBOASG %P 2:A194 = EIN, 3: BOASG
         $OUT[194] = TRUE
      ;ENDFOLD
      ;FOLD -- Quitt. Fraesen SK3 AUS -- ;%{SE}%MKUKATPVW %CVW_COM %VCOMMENT %P 2:-- Quitt. Fraesen SK3 AUS --, 3: VW_COMMENT
      ;ENDFOLD
      ;FOLD A1106 = F832 & A1106 ;%{SE}%MKUKATPVW %CVW_SPS %VBOASG %P 2:A1106 = F832 & A1106, 3: BOASG
         $OUT[1106] = $FLAG[832] AND $OUT[1106]
      ;ENDFOLD
      ;FOLD A1042 = !F832 & A1042 ;%{SE}%MKUKATPVW %CVW_SPS %VBOASG %P 2:A1042 = !F832 & A1042, 3: BOASG
         $OUT[1042] = NOT $FLAG[832] AND $OUT[1042]
      ;ENDFOLD
      ;FOLD Schritt 98 = T8 & A4039  ;%{SE}%MKUKATPVW %CVW_SPS %VST_CON %P 2:Schritt 98 = T8 & A4039 , 3: ST_CON
         IF $TIMER_FLAG[8] AND $OUT[4039] THEN
            PREVSTEP = $APP_INT[5]
            $APP_INT[5] = 98
         ENDIF
      ;ENDFOLD
   ;ENDFOLD
   ;FOLD SCHRITT 98 -- STAT EZ3/SP3/KE3 -- ;%{P}%MKUKATPVW,%CSTEP,%VST_NR,%P 1:SCHRITT, 2:98, 3: STAT EZ3/SP3/KE3
      ;FOLD ;%{H}
         Case 98
      ;ENDFOLD
      ;FOLD -- Hilfsflag SK Programmwechsel -- ;%{SE}%MKUKATPVW %CVW_COM %VCOMMENT %P 2:-- Hilfsflag SK Programmwechsel --, 3: VW_COMMENT
      ;ENDFOLD
      ;FOLD F334 = AUS ;%{SE}%MKUKATPVW %CVW_SPS %VBOASG %P 2:F334 = AUS, 3: BOASG
         $FLAG[334] = FALSE
      ;ENDFOLD
      ;FOLD -- Ueberwachungszeit KF3 EIN -- ;%{SE}%MKUKATPVW %CVW_COM %VCOMMENT %P 2:-- Ueberwachungszeit KF3 EIN --, 3: VW_COMMENT
      ;ENDFOLD
      ;FOLD T7 ( EIN ) = -30[1/10Sek] ;%{SE}%MKUKATPVW %CVW_SPS %VTASG %P 2:T7 ( EIN ) = -30[1/10Sek], 3: TASG
         VW(#SET_TIME,TRUE,7,0,-30)
      ;ENDFOLD
      ;FOLD -- KF3 einschalten -- ;%{SE}%MKUKATPVW %CVW_COM %VCOMMENT %P 2:-- KF3 einschalten --, 3: VW_COMMENT
      ;ENDFOLD
      ;FOLD i1 (EIN) = 0 ;%{SE}%MKUKATPVW %CVW_SPS %VARIASG %P 2:i1 (EIN) = 0, 3: ARIASG
         VW(#COUNTER,TRUE,1,0)
      ;ENDFOLD
      ;FOLD A1154 = EIN ;%{SE}%MKUKATPVW %CVW_SPS %VBOASG %P 2:A1154 = EIN, 3: BOASG
         $OUT[1154] = TRUE
      ;ENDFOLD
      ;FOLD Schritt 99 = A4039  ;%{SE}%MKUKATPVW %CVW_SPS %VST_CON %P 2:Schritt 99 = A4039 , 3: ST_CON
         IF $OUT[4039] THEN
            PREVSTEP = $APP_INT[5]
            $APP_INT[5] = 99
         ENDIF
      ;ENDFOLD
   ;ENDFOLD
   ;FOLD SCHRITT 99 -- STAT EZ3/SP3/KE3 -- ;%{P}%MKUKATPVW,%CSTEP,%VST_NR,%P 1:SCHRITT, 2:99, 3: STAT EZ3/SP3/KE3
      ;FOLD ;%{H}
         Case 99
      ;ENDFOLD
      ;FOLD -- Funktionstest KF Motor -- ;%{SE}%MKUKATPVW %CVW_COM %VCOMMENT %P 2:-- Funktionstest KF Motor --, 3: VW_COMMENT
      ;ENDFOLD
      ;FOLD F312 = EIN ;%{SE}%MKUKATPVW %CVW_SPS %VBOASG %P 2:F312 = EIN, 3: BOASG
         $FLAG[312] = TRUE
      ;ENDFOLD
      ;FOLD F313 = i1 > 2 ;%{SE}%MKUKATPVW %CVW_SPS %VBOCMP %P 2:F313 = i1 > 2, 3: BOCMP
         $FLAG[313] = $COUNT_I[1] > 2
      ;ENDFOLD
      ;FOLD Schritt 100 = (F313 + T7) & A4039  ;%{SE}%MKUKATPVW %CVW_SPS %VST_CON %P 2:Schritt 100 = (F313 + T7) & A4039 , 3: ST_CON
         IF ($FLAG[313] OR $TIMER_FLAG[7]) AND $OUT[4039] THEN
            PREVSTEP = $APP_INT[5]
            $APP_INT[5] = 100
         ENDIF
      ;ENDFOLD
   ;ENDFOLD
   ;FOLD SCHRITT 100 -- STAT EZ3/SP3/KE3 -- ;%{P}%MKUKATPVW,%CSTEP,%VST_NR,%P 1:SCHRITT, 2:100, 3: STAT EZ3/SP3/KE3
      ;FOLD ;%{H}
         Case 100
      ;ENDFOLD
      ;FOLD F312 = AUS ;%{SE}%MKUKATPVW %CVW_SPS %VBOASG %P 2:F312 = AUS, 3: BOASG
         $FLAG[312] = FALSE
      ;ENDFOLD
      ;FOLD -- Ueberwachungszeit KS3 schwenken -- ;%{SE}%MKUKATPVW %CVW_COM %VCOMMENT %P 2:-- Ueberwachungszeit KS3 schwenken --, 3: VW_COMMENT
      ;ENDFOLD
      ;FOLD t8 ( EIN ) = -100[1/10Sek] ;%{SE}%MKUKATPVW %CVW_SPS %VTASG %P 2:t8 ( EIN ) = -100[1/10Sek], 3: TASG
         VW(#SET_TIME,TRUE,8,0,-100)
      ;ENDFOLD
      ;FOLD Schritt 101 = A4039  ;%{SE}%MKUKATPVW %CVW_SPS %VST_CON %P 2:Schritt 101 = A4039 , 3: ST_CON
         IF $OUT[4039] THEN
            PREVSTEP = $APP_INT[5]
            $APP_INT[5] = 101
         ENDIF
      ;ENDFOLD
   ;ENDFOLD
   ;FOLD SCHRITT 101 -- STAT EZ3/SP3/KE3 -- ;%{P}%MKUKATPVW,%CSTEP,%VST_NR,%P 1:SCHRITT, 2:101, 3: STAT EZ3/SP3/KE3
      ;FOLD ;%{H}
         Case 101
      ;ENDFOLD
      ;FOLD -- RSK Fehlerausgabe KF1 Initiator/Motor -- ;%{SE}%MKUKATPVW %CVW_COM %VCOMMENT %P 2:-- RSK Fehlerausgabe KF1 Initiator/Motor --, 3: VW_COMMENT
      ;ENDFOLD
      ;FOLD F322 = !F313 ;%{SE}%MKUKATPVW %CVW_SPS %VBOASG %P 2:F322 = !F313, 3: BOASG
         $FLAG[322] = NOT $FLAG[313]
      ;ENDFOLD
      ;FOLD -- RSK Fehlerausgabe KS3 Ruhest. -- ;%{SE}%MKUKATPVW %CVW_COM %VCOMMENT %P 2:-- RSK Fehlerausgabe KS3 Ruhest. --, 3: VW_COMMENT
      ;ENDFOLD
      ;FOLD F323 = (!E1162 + E1163 + E1164 + !E1165) & !F324 & !F328 ;%{SE}%MKUKATPVW %CVW_SPS %VBOASG %P 2:F323 = (!E1162 + E1163 + E1164 + !E1165) & !F324 & !F328, 3: BOASG
         $FLAG[323] = (NOT $IN[1162] OR $IN[1163] OR $IN[1164] OR NOT $IN[1165]) AND NOT $FLAG[324] AND NOT $FLAG[328]
      ;ENDFOLD
      ;FOLD -- RSK Sammelstoerung -- ;%{SE}%MKUKATPVW %CVW_COM %VCOMMENT %P 2:-- RSK Sammelstoerung --, 3: VW_COMMENT
      ;ENDFOLD
      ;FOLD F329 = F322 + F323 ;%{SE}%MKUKATPVW %CVW_SPS %VBOASG %P 2:F329 = F322 + F323, 3: BOASG
         $FLAG[329] = $FLAG[322] OR $FLAG[323]
      ;ENDFOLD
      ;FOLD T7 ( EIN ) = STOP ;%{SE}%MKUKATPVW %CVW_SPS %VTSTOP %P 2:T7 ( EIN ) = STOP, 3: TSTOP
         VW(#SET_TIME,TRUE,7,1,0)
      ;ENDFOLD
      ;FOLD A1154 = !F322 & !F323 ;%{SE}%MKUKATPVW %CVW_SPS %VBOASG %P 2:A1154 = !F322 & !F323, 3: BOASG
         $OUT[1154] = NOT $FLAG[322] AND NOT $FLAG[323]
      ;ENDFOLD
      ;FOLD -- KF3 Versetzeinheit vor -- ;%{SE}%MKUKATPVW %CVW_COM %VCOMMENT %P 2:-- KF3 Versetzeinheit vor --, 3: VW_COMMENT
      ;ENDFOLD
      ;FOLD A1155 = !F322 & !F323 & F564 ;%{SE}%MKUKATPVW %CVW_SPS %VBOASG %P 2:A1155 = !F322 & !F323 & F564, 3: BOASG
         $OUT[1155] = NOT $FLAG[322] AND NOT $FLAG[323] AND $FLAG[564]
      ;ENDFOLD
      ;FOLD Schritt 102 = (!F322 & !F323 & (E1155 & F564 + !E1155 & !F564) + T8) & A4039  ;%{SE}%MKUKATPVW %CVW_SPS %VST_CON %P 2:Schritt 102 = (!F322 & !F323 & (E1155 & F564 + !E1155 & !F564) + T8) & A4039 , 3: ST_CON
         IF (NOT $FLAG[322] AND NOT $FLAG[323] AND ($IN[1155] AND $FLAG[564] OR NOT $IN[1155] AND NOT $FLAG[564]) OR $TIMER_FLAG[8]) AND $OUT[4039] THEN
            PREVSTEP = $APP_INT[5]
            $APP_INT[5] = 102
         ENDIF
      ;ENDFOLD
      ;FOLD Schritt 118 = (F322 + F323) & !F324 & !F328 & A4039  ;%{SE}%MKUKATPVW %CVW_SPS %VST_CON %P 2:Schritt 118 = (F322 + F323) & !F324 & !F328 & A4039 , 3: ST_CON
         IF ($FLAG[322] OR $FLAG[323]) AND NOT $FLAG[324] AND NOT $FLAG[328] AND $OUT[4039] THEN
            PREVSTEP = $APP_INT[5]
            $APP_INT[5] = 118
         ENDIF
      ;ENDFOLD
   ;ENDFOLD
   ;FOLD SCHRITT 102 -- STAT EZ3/SP3/KE3 -- ;%{P}%MKUKATPVW,%CSTEP,%VST_NR,%P 1:SCHRITT, 2:102, 3: STAT EZ3/SP3/KE3
      ;FOLD ;%{H}
         Case 102
      ;ENDFOLD
      ;FOLD F329 = T8 ;%{SE}%MKUKATPVW %CVW_SPS %VBOASG %P 2:F329 = T8, 3: BOASG
         $FLAG[329] = $TIMER_FLAG[8]
      ;ENDFOLD
      ;FOLD F324 = AUS ;%{SE}%MKUKATPVW %CVW_SPS %VBOASG %P 2:F324 = AUS, 3: BOASG
         $FLAG[324] = FALSE
      ;ENDFOLD
      ;FOLD F328 = AUS ;%{SE}%MKUKATPVW %CVW_SPS %VBOASG %P 2:F328 = AUS, 3: BOASG
         $FLAG[328] = FALSE
      ;ENDFOLD
      ;FOLD -- KS3 in Arbeitsstellung schwenken -- ;%{SE}%MKUKATPVW %CVW_COM %VCOMMENT %P 2:-- KS3 in Arbeitsstellung schwenken --, 3: VW_COMMENT
      ;ENDFOLD
      ;FOLD A1162 = (F747 + !F714) & (E1037 + F714) & !E1163 & (E1155 & F564 + !E1155 & !F564) ;%{SE}%MKUKATPVW %CVW_SPS %VBOASG %P 2:A1162 = (F747 + !F714) & (E1037 + F714) & !E1163 & (E1155 & F564 + !E1155 & !F564), 3: BOASG
         $OUT[1162] = ($FLAG[747] OR NOT $FLAG[714]) AND ($IN[1037] OR $FLAG[714]) AND NOT $IN[1163] AND ($IN[1155] AND $FLAG[564] OR NOT $IN[1155] AND NOT $FLAG[564])
      ;ENDFOLD
      ;FOLD -- KF3 Ausblasen -- ;%{SE}%MKUKATPVW %CVW_COM %VCOMMENT %P 2:-- KF3 Ausblasen --, 3: VW_COMMENT
      ;ENDFOLD
      ;FOLD A1167 = F330 + !F330 & !F331 & !F332 ;%{SE}%MKUKATPVW %CVW_SPS %VBOASG %P 2:A1167 = F330 + !F330 & !F331 & !F332, 3: BOASG
         $OUT[1167] = $FLAG[330] OR NOT $FLAG[330] AND NOT $FLAG[331] AND NOT $FLAG[332]
      ;ENDFOLD
      ;FOLD Schritt 103 = (F747 + !F714) & (E1037 + F714) & (A1162 + E1163 + T8) & A4039  ;%{SE}%MKUKATPVW %CVW_SPS %VST_CON %P 2:Schritt 103 = (F747 + !F714) & (E1037 + F714) & (A1162 + E1163 + T8) & A4039 , 3: ST_CON
         IF ($FLAG[747] OR NOT $FLAG[714]) AND ($IN[1037] OR $FLAG[714]) AND ($OUT[1162] OR $IN[1163] OR $TIMER_FLAG[8]) AND $OUT[4039] THEN
            PREVSTEP = $APP_INT[5]
            $APP_INT[5] = 103
         ENDIF
      ;ENDFOLD
   ;ENDFOLD
   ;FOLD SCHRITT 103 -- STAT EZ3/SP3/KE3 -- ;%{P}%MKUKATPVW,%CSTEP,%VST_NR,%P 1:SCHRITT, 2:103, 3: STAT EZ3/SP3/KE3
      ;FOLD ;%{H}
         Case 103
      ;ENDFOLD
      ;FOLD -- RSK Fehlerausgabe KF Versetzeinheit -- ;%{SE}%MKUKATPVW %CVW_COM %VCOMMENT %P 2:-- RSK Fehlerausgabe KF Versetzeinheit --, 3: VW_COMMENT
      ;ENDFOLD
      ;FOLD F328 = !E1155 & F564 & !F324 ;%{SE}%MKUKATPVW %CVW_SPS %VBOASG %P 2:F328 = !E1155 & F564 & !F324, 3: BOASG
         $FLAG[328] = NOT $IN[1155] AND $FLAG[564] AND NOT $FLAG[324]
      ;ENDFOLD
      ;FOLD -- RSK Fehlerausgabe KS3 Arbeitsstellung -- ;%{SE}%MKUKATPVW %CVW_COM %VCOMMENT %P 2:-- RSK Fehlerausgabe KS3 Arbeitsstellung --, 3: VW_COMMENT
      ;ENDFOLD
      ;FOLD F324 = (E1162 + !E1163 + !E1164 + E1165) & T8 & (E1155 + !F564) + F324 ;%{SE}%MKUKATPVW %CVW_SPS %VBOASG %P 2:F324 = (E1162 + !E1163 + !E1164 + E1165) & T8 & (E1155 + !F564) + F324, 3: BOASG
         $FLAG[324] = ($IN[1162] OR NOT $IN[1163] OR NOT $IN[1164] OR $IN[1165]) AND $TIMER_FLAG[8] AND ($IN[1155] OR NOT $FLAG[564]) OR $FLAG[324]
      ;ENDFOLD
      ;FOLD -- RSK Fehlerausgabe EZ/SP min. Oeffnung -- ;%{SE}%MKUKATPVW %CVW_COM %VCOMMENT %P 2:-- RSK Fehlerausgabe EZ/SP min. Oeffnung --, 3: VW_COMMENT
      ;ENDFOLD
      ;FOLD F333 = !F747 ;%{SE}%MKUKATPVW %CVW_SPS %VBOASG %P 2:F333 = !F747, 3: BOASG
         $FLAG[333] = NOT $FLAG[747]
      ;ENDFOLD
      ;FOLD -- RSK Sammelstoerung -- ;%{SE}%MKUKATPVW %CVW_COM %VCOMMENT %P 2:-- RSK Sammelstoerung --, 3: VW_COMMENT
      ;ENDFOLD
      ;FOLD F329 = F324 + F328 ;%{SE}%MKUKATPVW %CVW_SPS %VBOASG %P 2:F329 = F324 + F328, 3: BOASG
         $FLAG[329] = $FLAG[324] OR $FLAG[328]
      ;ENDFOLD
      ;FOLD A1154 = !F324 & !F328 ;%{SE}%MKUKATPVW %CVW_SPS %VBOASG %P 2:A1154 = !F324 & !F328, 3: BOASG
         $OUT[1154] = NOT $FLAG[324] AND NOT $FLAG[328]
      ;ENDFOLD
      ;FOLD -- KF3 Ausblasen -- ;%{SE}%MKUKATPVW %CVW_COM %VCOMMENT %P 2:-- KF3 Ausblasen --, 3: VW_COMMENT
      ;ENDFOLD
      ;FOLD A1167 = (F330 + !F330 & !F331 & !F332) & !F324 & !F328 ;%{SE}%MKUKATPVW %CVW_SPS %VBOASG %P 2:A1167 = (F330 + !F330 & !F331 & !F332) & !F324 & !F328, 3: BOASG
         $OUT[1167] = ($FLAG[330] OR NOT $FLAG[330] AND NOT $FLAG[331] AND NOT $FLAG[332]) AND NOT $FLAG[324] AND NOT $FLAG[328]
      ;ENDFOLD
      ;FOLD A1155 = F564 ;%{SE}%MKUKATPVW %CVW_SPS %VBOASG %P 2:A1155 = F564, 3: BOASG
         $OUT[1155] = $FLAG[564]
      ;ENDFOLD
      ;FOLD -- Ueberwachungszeit EZ3/SP3/KE3 schliessen -- ;%{SE}%MKUKATPVW %CVW_COM %VCOMMENT %P 2:-- Ueberwachungszeit EZ3/SP3/KE3 schliessen --, 3: VW_COMMENT
      ;ENDFOLD
      ;FOLD t9 ( EIN ) = -100[1/10Sek] ;%{SE}%MKUKATPVW %CVW_SPS %VTASG %P 2:t9 ( EIN ) = -100[1/10Sek], 3: TASG
         VW(#SET_TIME,TRUE,9,0,-100)
      ;ENDFOLD
      ;FOLD -- Verweilzeit Versetzeinheit Rueck -- ;%{SE}%MKUKATPVW %CVW_COM %VCOMMENT %P 2:-- Verweilzeit Versetzeinheit Rueck --, 3: VW_COMMENT
      ;ENDFOLD
      ;FOLD t11 ( EIN ) = i24[1/10Sek] ;%{SE}%MKUKATPVW %CVW_SPS %VTASG %P 2:t11 ( EIN ) = i24[1/10Sek], 3: TASG
         VW(#SET_TIME,TRUE,11,0,$COUNT_I[24])
      ;ENDFOLD
      ;FOLD Schritt 98 = (F324 + F328) & (E26 + E27) & A4039  ;%{SE}%MKUKATPVW %CVW_SPS %VST_CON %P 2:Schritt 98 = (F324 + F328) & (E26 + E27) & A4039 , 3: ST_CON
         IF ($FLAG[324] OR $FLAG[328]) AND ($IN[26] OR $IN[27]) AND $OUT[4039] THEN
            PREVSTEP = $APP_INT[5]
            $APP_INT[5] = 98
         ENDIF
      ;ENDFOLD
      ;FOLD Schritt 104 = !F324 & !F328 & !E1162 & E1163 & E1164 & !E1165 & A4039  ;%{SE}%MKUKATPVW %CVW_SPS %VST_CON %P 2:Schritt 104 = !F324 & !F328 & !E1162 & E1163 & E1164 & !E1165 & A4039 , 3: ST_CON
         IF NOT $FLAG[324] AND NOT $FLAG[328] AND NOT $IN[1162] AND $IN[1163] AND $IN[1164] AND NOT $IN[1165] AND $OUT[4039] THEN
            PREVSTEP = $APP_INT[5]
            $APP_INT[5] = 104
         ENDIF
      ;ENDFOLD
   ;ENDFOLD
   ;FOLD SCHRITT 104 -- STAT EZ3/SP3/KE3 -- ;%{P}%MKUKATPVW,%CSTEP,%VST_NR,%P 1:SCHRITT, 2:104, 3: STAT EZ3/SP3/KE3
      ;FOLD ;%{H}
         Case 104
      ;ENDFOLD
      ;FOLD -- Umdreh. KF setzen -- ;%{SE}%MKUKATPVW %CVW_COM %VCOMMENT %P 2:-- Umdreh. KF setzen --, 3: VW_COMMENT
      ;ENDFOLD
      ;FOLD F270 = F191 & F732 ;%{SE}%MKUKATPVW %CVW_SPS %VBOASG %P 2:F270 = F191 & F732, 3: BOASG
         $FLAG[270] = $FLAG[191] AND $FLAG[732]
      ;ENDFOLD
      ;FOLD i45 ( EIN ) = i19 ;%{SE}%MKUKATPVW %CVW_SPS %VARIASG %P 2:i45 ( EIN ) = i19, 3: ARIASG
         VW(#COUNTER,TRUE,45,$COUNT_I[19])
      ;ENDFOLD
      ;FOLD i19 ( F270 ) = i38 ;%{SE}%MKUKATPVW %CVW_SPS %VARIASG %P 2:i19 ( F270 ) = i38, 3: ARIASG
         VW(#COUNTER,$FLAG[270],19,$COUNT_I[38])
      ;ENDFOLD
      ;FOLD i1 ( EIN ) = 0 ;%{SE}%MKUKATPVW %CVW_SPS %VARIASG %P 2:i1 ( EIN ) = 0, 3: ARIASG
         VW(#COUNTER,TRUE,1,0)
      ;ENDFOLD
      ;FOLD F190 = AUS ;%{SE}%MKUKATPVW %CVW_SPS %VBOASG %P 2:F190 = AUS, 3: BOASG
         $FLAG[190] = FALSE
      ;ENDFOLD
      ;FOLD F312 = AUS ;%{SE}%MKUKATPVW %CVW_SPS %VBOASG %P 2:F312 = AUS, 3: BOASG
         $FLAG[312] = FALSE
      ;ENDFOLD
      ;FOLD F313 = AUS ;%{SE}%MKUKATPVW %CVW_SPS %VBOASG %P 2:F313 = AUS, 3: BOASG
         $FLAG[313] = FALSE
      ;ENDFOLD
      ;FOLD F324 = AUS ;%{SE}%MKUKATPVW %CVW_SPS %VBOASG %P 2:F324 = AUS, 3: BOASG
         $FLAG[324] = FALSE
      ;ENDFOLD
      ;FOLD F328 = AUS ;%{SE}%MKUKATPVW %CVW_SPS %VBOASG %P 2:F328 = AUS, 3: BOASG
         $FLAG[328] = FALSE
      ;ENDFOLD
      ;FOLD -- KF3 einschalten nach Fehler -- ;%{SE}%MKUKATPVW %CVW_COM %VCOMMENT %P 2:-- KF3 einschalten nach Fehler --, 3: VW_COMMENT
      ;ENDFOLD
      ;FOLD A1154 = EIN ;%{SE}%MKUKATPVW %CVW_SPS %VBOASG %P 2:A1154 = EIN, 3: BOASG
         $OUT[1154] = TRUE
      ;ENDFOLD
      ;FOLD -- KF3 Versetzeinheit rueck -- ;%{SE}%MKUKATPVW %CVW_COM %VCOMMENT %P 2:-- KF3 Versetzeinheit rueck --, 3: VW_COMMENT
      ;ENDFOLD
      ;FOLD A1155 = AUS ;%{SE}%MKUKATPVW %CVW_SPS %VBOASG %P 2:A1155 = AUS, 3: BOASG
         $OUT[1155] = FALSE
      ;ENDFOLD
      ;FOLD Schritt 105 = T11 & A4039  ;%{SE}%MKUKATPVW %CVW_SPS %VST_CON %P 2:Schritt 105 = T11 & A4039 , 3: ST_CON
         IF $TIMER_FLAG[11] AND $OUT[4039] THEN
            PREVSTEP = $APP_INT[5]
            $APP_INT[5] = 105
         ENDIF
      ;ENDFOLD
   ;ENDFOLD
   ;FOLD SCHRITT 105 -- STAT EZ3/SP3/KE3 -- ;%{P}%MKUKATPVW,%CSTEP,%VST_NR,%P 1:SCHRITT, 2:105, 3: STAT EZ3/SP3/KE3
      ;FOLD ;%{H}
         Case 105
      ;ENDFOLD
      ;FOLD F270 = AUS ;%{SE}%MKUKATPVW %CVW_SPS %VBOASG %P 2:F270 = AUS, 3: BOASG
         $FLAG[270] = FALSE
      ;ENDFOLD
      ;FOLD t11 ( EIN ) = STOP ;%{SE}%MKUKATPVW %CVW_SPS %VTSTOP %P 2:t11 ( EIN ) = STOP, 3: TSTOP
         VW(#SET_TIME,TRUE,11,1,0)
      ;ENDFOLD
      ;FOLD -- EZ3/SP3/KE3 schliessen -- ;%{SE}%MKUKATPVW %CVW_COM %VCOMMENT %P 2:-- EZ3/SP3/KE3 schliessen --, 3: VW_COMMENT
      ;ENDFOLD
      ;FOLD A1037 = AUS ;%{SE}%MKUKATPVW %CVW_SPS %VBOASG %P 2:A1037 = AUS, 3: BOASG
         $OUT[1037] = FALSE
      ;ENDFOLD
      ;FOLD A1038 = EIN ;%{SE}%MKUKATPVW %CVW_SPS %VBOASG %P 2:A1038 = EIN, 3: BOASG
         $OUT[1038] = TRUE
      ;ENDFOLD
      ;FOLD -- KF3 Ausblasen -- ;%{SE}%MKUKATPVW %CVW_COM %VCOMMENT %P 2:-- KF3 Ausblasen --, 3: VW_COMMENT
      ;ENDFOLD
      ;FOLD A1167 = F330 + F331 + !F330 & !F331 & !F332 ;%{SE}%MKUKATPVW %CVW_SPS %VBOASG %P 2:A1167 = F330 + F331 + !F330 & !F331 & !F332, 3: BOASG
         $OUT[1167] = $FLAG[330] OR $FLAG[331] OR NOT $FLAG[330] AND NOT $FLAG[331] AND NOT $FLAG[332]
      ;ENDFOLD
      ;FOLD Schritt 106 = (!E1037 & E1038 + T9) & A4039  ;%{SE}%MKUKATPVW %CVW_SPS %VST_CON %P 2:Schritt 106 = (!E1037 & E1038 + T9) & A4039 , 3: ST_CON
         IF (NOT $IN[1037] AND $IN[1038] OR $TIMER_FLAG[9]) AND $OUT[4039] THEN
            PREVSTEP = $APP_INT[5]
            $APP_INT[5] = 106
         ENDIF
      ;ENDFOLD
   ;ENDFOLD
   ;FOLD SCHRITT 106 -- STAT EZ3/SP3/KE3 -- ;%{P}%MKUKATPVW,%CSTEP,%VST_NR,%P 1:SCHRITT, 2:106, 3: STAT EZ3/SP3/KE3
      ;FOLD ;%{H}
         Case 106
      ;ENDFOLD
      ;FOLD -- RSK Fehlerausgabe Kraftaufbau -- ;%{SE}%MKUKATPVW %CVW_COM %VCOMMENT %P 2:-- RSK Fehlerausgabe Kraftaufbau --, 3: VW_COMMENT
      ;ENDFOLD
      ;FOLD F325 = T9 ;%{SE}%MKUKATPVW %CVW_SPS %VBOASG %P 2:F325 = T9, 3: BOASG
         $FLAG[325] = $TIMER_FLAG[9]
      ;ENDFOLD
      ;FOLD -- RSK Sammelstoerung -- ;%{SE}%MKUKATPVW %CVW_COM %VCOMMENT %P 2:-- RSK Sammelstoerung --, 3: VW_COMMENT
      ;ENDFOLD
      ;FOLD F329 = F325 ;%{SE}%MKUKATPVW %CVW_SPS %VBOASG %P 2:F329 = F325, 3: BOASG
         $FLAG[329] = $FLAG[325]
      ;ENDFOLD
      ;FOLD -- KF3 abschalten bei Fehler -- ;%{SE}%MKUKATPVW %CVW_COM %VCOMMENT %P 2:-- KF3 abschalten bei Fehler --, 3: VW_COMMENT
      ;ENDFOLD
      ;FOLD A1154 = !T9 ;%{SE}%MKUKATPVW %CVW_SPS %VBOASG %P 2:A1154 = !T9, 3: BOASG
         $OUT[1154] = NOT $TIMER_FLAG[9]
      ;ENDFOLD
      ;FOLD -- KF3 Ausblasen -- ;%{SE}%MKUKATPVW %CVW_COM %VCOMMENT %P 2:-- KF3 Ausblasen --, 3: VW_COMMENT
      ;ENDFOLD
      ;FOLD A1167 = (F330 + F331 + !F330 & !F331 & !F332) & !T9 ;%{SE}%MKUKATPVW %CVW_SPS %VBOASG %P 2:A1167 = (F330 + F331 + !F330 & !F331 & !F332) & !T9, 3: BOASG
